   1:  PR[91,2] = PR[90,2] + 13.774;
   1:L PR[91] R[100]mm/sec CNT100;
   1:  PR[91,1] = PR[90,1] + 28.237;
   1:  PR[91,2] = PR[90,2] + 15.206;
   1:L PR[91] R[100]mm/sec CNT100;
   1:  PR[91,1] = PR[90,1] + 27.710;
   1:  PR[91,2] = PR[90,2] + 15.533;
   1:L PR[91] R[100]mm/sec CNT100;
   1:  PR[91,1] = PR[90,1] + 25.602;
   1:  PR[91,2] = PR[90,2] + 16.678;
   1:L PR[91] R[100]mm/sec CNT100;
   1:  PR[91,1] = PR[90,1] + 23.587;
   1:  PR[91,2] = PR[90,2] + 17.443;
   1:L PR[91] R[100]mm/sec CNT100;
   1:  PR[91,1] = PR[90,1] + 22.466;
   1:  PR[91,2] = PR[90,2] + 17.845;
   1:L PR[91] R[100]mm/sec CNT100;
   1:  PR[91,1] = PR[90,1] + 20.601;
   1:  PR[91,2] = PR[90,2] + 18.286;
   1:L PR[91] R[100]mm/sec CNT100;
   1:  PR[91,1] = PR[90,1] + 18.780;
   1:  PR[91,2] = PR[90,2] + 18.458;
   1:L PR[91] R[100]mm/sec CNT100;
   1:  PR[91,1] = PR[90,1] + 17.067;
   1:  PR[91,2] = PR[90,2] + 18.689;
   1:L PR[91] R[100]mm/sec CNT100;
   1:  PR[91,1] = PR[90,1] + 15.509;
   1:  PR[91,2] = PR[90,2] + 18.636;
   1:L PR[91] R[100]mm/sec CNT100;
   1:  PR[91,1] = PR[90,1] + 13.386;
   1:  PR[91,2] = PR[90,2] + 18.465;
   1:L PR[91] R[100]mm/sec CNT100;
   1:  PR[91,1] = PR[90,1] + 12.007;
   1:  PR[91,2] = PR[90,2] + 18.232;
   1:L PR[91] R[100]mm/sec CNT100;
   1:  PR[91,1] = PR[90,1] + 10.743;
   1:  PR[91,2] = PR[90,2] + 17.834;
   1:L PR[91] R[100]mm/sec CNT100;
   1:  PR[91,1] = PR[90,1] + 8.282;
   1:  PR[91,2] = PR[90,2] + 17.090;
   1:L PR[91] R[100]mm/sec CNT100;
   1:  PR[91,1] = PR[90,1] + 7.321;
   1:  PR[91,2] = PR[90,2] + 16.639;
   1:L PR[91] R[100]mm/sec CNT100;
   1:  PR[91,1] = PR[90,1] + 4.764;
   1:  PR[91,2] = PR[90,2] + 15.203;
   1:L PR[91] R[100]mm/sec CNT100;
   1:  PR[91,1] = PR[90,1] + 3.982;
   1:  PR[91,2] = PR[90,2] + 14.693;
   1:L PR[91] R[100]mm/sec CNT100;
   1:  PR[91,1] = PR[90,1] + 2.880;
   1:  PR[91,2] = PR[90,2] + 13.777;
   1:L PR[91] R[100]mm/sec CNT100;
   1:  PR[91,1] = PR[90,1] + 2.134;
   1:  PR[91,2] = PR[90,2] + 13.086;
   1:L PR[91] R[100]mm/sec CNT100;
   1:  PR[91,1] = PR[90,1] + 1.372;
   1:  PR[91,2] = PR[90,2] + 12.629;
   1:L PR[91] R[100]mm/sec CNT100;
   1:  PR[91,1] = PR[90,1] + 0.512;
   1:  PR[91,2] = PR[90,2] + 12.269;
   1:L PR[91] R[100]mm/sec CNT100;
   1:  PR[91] = PR[90];
   1:  PR[91,1] = PR[90,1] + -1.049;
   1:  PR[91,2] = PR[90,2] + 12.856;
   1:  PR[91,3] = PR[90,3] + 32.695;
   1:L PR[91] R[100]mm/sec CNT100;
   1:  PR[91,1] = PR[90,1] + -2.250;
   1:  PR[91,2] = PR[90,2] + 13.413;
   1:L PR[91] R[100]mm/sec CNT100;
   1:  PR[91,1] = PR[90,1] + -3.926;
   1:  PR[91,2] = PR[90,2] + 14.817;
   1:L PR[91] R[100]mm/sec CNT100;
   1:  PR[91,1] = PR[90,1] + -4.466;
   1:  PR[91,2] = PR[90,2] + 15.172;
   1:L PR[91] R[100]mm/sec CNT100;
   1:  PR[91,1] = PR[90,1] + -7.479;
   1:  PR[91,2] = PR[90,2] + 16.866;
   1:L PR[91] R[100]mm/sec CNT100;
   1:  PR[91,1] = PR[90,1] + -8.163;
   1:  PR[91,2] = PR[90,2] + 17.188;
   1:L PR[91] R[100]mm/sec CNT100;
   1:  PR[91,1] = PR[90,1] + -12.073;
   1:  PR[91,2] = PR[90,2] + 18.383;
   1:L PR[91] R[100]mm/sec CNT100;
   1:  PR[91,1] = PR[90,1] + -13.127;
   1:  PR[91,2] = PR[90,2] + 18.559;
   1:L PR[91] R[100]mm/sec CNT100;
   1:  PR[91,1] = PR[90,1] + -15.795;
   1:  PR[91,2] = PR[90,2] + 18.773;
   1:L PR[91] R[100]mm/sec CNT100;
   1:  PR[91,1] = PR[90,1] + -17.081;
   1:  PR[91,2] = PR[90,2] + 18.816;
   1:L PR[91] R[100]mm/sec CNT100;
   1:  PR[91,1] = PR[90,1] + -18.591;
   1:  PR[91,2] = PR[90,2] + 18.666;
   1:L PR[91] R[100]mm/sec CNT100;
   1:  PR[91,1] = PR[90,1] + -20.751;
   1:  PR[91,2] = PR[90,2] + 18.379;
   1:L PR[91] R[100]mm/sec CNT100;
   1:  PR[91,1] = PR[90,1] + -22.305;
   1:  PR[91,2] = PR[90,2] + 18.011;
   1:L PR[91] R[100]mm/sec CNT100;
   1:  PR[91,1] = PR[90,1] + -24.173;
   1:  PR[91,2] = PR[90,2] + 17.302;
   1:L PR[91] R[100]mm/sec CNT100;
   1:  PR[91,1] = PR[90,1] + -25.691;
   1:  PR[91,2] = PR[90,2] + 16.756;
   1:L PR[91] R[100]mm/sec CNT100;
   1:  PR[91,1] = PR[90,1] + -27.462;
   1:  PR[91,2] = PR[90,2] + 15.788;
   1:L PR[91] R[100]mm/sec CNT100;
   1:  PR[91,1] = PR[90,1] + -28.488;
   1:  PR[91,2] = PR[90,2] + 15.149;
   1:L PR[91] R[100]mm/sec CNT100;
   1:  PR[91,1] = PR[90,1] + -30.178;
   1:  PR[91,2] = PR[90,2] + 13.903;
   1:L PR[91] R[100]mm/sec CNT100;
   1:  PR[91,1] = PR[90,1] + -32.399;
   1:  PR[91,2] = PR[90,2] + 11.739;
   1:L PR[91] R[100]mm/sec CNT100;
   1:  PR[91,1] = PR[90,1] + -33.837;
   1:  PR[91,2] = PR[90,2] + 9.866;
   1:L PR[91] R[100]mm/sec CNT100;
   1:  PR[91,1] = PR[90,1] + -34.082;
   1:  PR[91,2] = PR[90,2] + 9.483;
   1:L PR[91] R[100]mm/sec CNT100;
   1:  PR[91,1] = PR[90,1] + -35.313;
   1:  PR[91,2] = PR[90,2] + 7.290;
   1:L PR[91] R[100]mm/sec CNT100;
   1:  PR[91,1] = PR[90,1] + -36.348;
   1:  PR[91,2] = PR[90,2] + 4.612;
   1:L PR[91] R[100]mm/sec CNT100;
   1:  PR[91,1] = PR[90,1] + -36.871;
   1:  PR[91,2] = PR[90,2] + 2.281;
   1:L PR[91] R[100]mm/sec CNT100;
   1:  PR[91,1] = PR[90,1] + -37.069;
   1:  PR[91,2] = PR[90,2] + -0.428;
   1:L PR[91] R[100]mm/sec CNT100;
   1:  PR[91,1] = PR[90,1] + -36.891;
   1:  PR[91,2] = PR[90,2] + -3.008;
   1:L PR[91] R[100]mm/sec CNT100;
   1:  PR[91,1] = PR[90,1] + -36.882;
   1:  PR[91,2] = PR[90,2] + -3.078;
   1:L PR[91] R[100]mm/sec CNT100;
   1:  PR[91,1] = PR[90,1] + -36.349;
   1:  PR[91,2] = PR[90,2] + -5.456;
   1:L PR[91] R[100]mm/sec CNT100;
   1:  PR[91,1] = PR[90,1] + -35.394;
   1:  PR[91,2] = PR[90,2] + -7.905;
   1:L PR[91] R[100]mm/sec CNT100;
   1:  PR[91,1] = PR[90,1] + -35.303;
   1:  PR[91,2] = PR[90,2] + -8.156;
   1:L PR[91] R[100]mm/sec CNT100;
   1:  PR[91,1] = PR[90,1] + -34.083;
   1:  PR[91,2] = PR[90,2] + -10.331;
   1:L PR[91] R[100]mm/sec CNT100;
   1:  PR[91,1] = PR[90,1] + -33.837;
   1:  PR[91,2] = PR[90,2] + -10.713;
   1:L PR[91] R[100]mm/sec CNT100;
   1:  PR[91,1] = PR[90,1] + -32.399;
   1:  PR[91,2] = PR[90,2] + -12.586;
   1:L PR[91] R[100]mm/sec CNT100;
   1:  PR[91,1] = PR[90,1] + -30.178;
   1:  PR[91,2] = PR[90,2] + -14.750;
   1:L PR[91] R[100]mm/sec CNT100;
   1:  PR[91,1] = PR[90,1] + -28.488;
   1:  PR[91,2] = PR[90,2] + -15.996;
   1:L PR[91] R[100]mm/sec CNT100;
   1:  PR[91,1] = PR[90,1] + -27.462;
   1:  PR[91,2] = PR[90,2] + -16.636;
   1:L PR[91] R[100]mm/sec CNT100;
   1:  PR[91,1] = PR[90,1] + -25.670;
   1:  PR[91,2] = PR[90,2] + -17.614;
   1:L PR[91] R[100]mm/sec CNT100;
   1:  PR[91,1] = PR[90,1] + -23.969;
   1:  PR[91,2] = PR[90,2] + -18.263;
   1:L PR[91] R[100]mm/sec CNT100;
   1:  PR[91,1] = PR[90,1] + -22.326;
   1:  PR[91,2] = PR[90,2] + -18.853;
   1:L PR[91] R[100]mm/sec CNT100;
   1:  PR[91,1] = PR[90,1] + -20.794;
   1:  PR[91,2] = PR[90,2] + -19.216;
   1:L PR[91] R[100]mm/sec CNT100;
   1:  PR[91,1] = PR[90,1] + -19.268;
   1:  PR[91,2] = PR[90,2] + -19.362;
   1:L PR[91] R[100]mm/sec CNT100;
   1:  PR[91,1] = PR[90,1] + -17.039;
   1:  PR[91,2] = PR[90,2] + -19.662;
   1:L PR[91] R[100]mm/sec CNT100;
   1:  PR[91,1] = PR[90,1] + -15.794;
   1:  PR[91,2] = PR[90,2] + -19.620;
   1:L PR[91] R[100]mm/sec CNT100;
   1:  PR[91,1] = PR[90,1] + -13.127;
   1:  PR[91,2] = PR[90,2] + -19.407;
   1:L PR[91] R[100]mm/sec CNT100;
   1:  PR[91,1] = PR[90,1] + -12.073;
   1:  PR[91,2] = PR[90,2] + -19.230;
   1:L PR[91] R[100]mm/sec CNT100;
   1:  PR[91,1] = PR[90,1] + -8.162;
   1:  PR[91,2] = PR[90,2] + -18.035;
   1:L PR[91] R[100]mm/sec CNT100;
   1:  PR[91,1] = PR[90,1] + -7.479;
   1:  PR[91,2] = PR[90,2] + -17.714;
   1:L PR[91] R[100]mm/sec CNT100;
   1:  PR[91,1] = PR[90,1] + -4.462;
   1:  PR[91,2] = PR[90,2] + -16.017;
   1:L PR[91] R[100]mm/sec CNT100;
   1:  PR[91,1] = PR[90,1] + -3.943;
   1:  PR[91,2] = PR[90,2] + -15.678;
   1:L PR[91] R[100]mm/sec CNT100;
   1:  PR[91,1] = PR[90,1] + -2.534;
   1:  PR[91,2] = PR[90,2] + -14.508;
   1:L PR[91] R[100]mm/sec CNT100;
   1:  PR[91,1] = PR[90,1] + -2.341;
   1:  PR[91,2] = PR[90,2] + -14.431;
   1:L PR[91] R[100]mm/sec CNT100;
   1:  PR[91,1] = PR[90,1] + -0.931;
   1:  PR[91,2] = PR[90,2] + -13.498;
   1:L PR[91] R[100]mm/sec CNT100;
   1:  PR[91,1] = PR[90,1] + 0.392;
   1:  PR[91,2] = PR[90,2] + -13.866;
   1:L PR[91] R[100]mm/sec CNT100;
   1:  PR[91,1] = PR[90,1] + 1.089;
   1:  PR[91,2] = PR[90,2] + -13.867;
   1:L PR[91] R[100]mm/sec CNT100;
   1:  PR[91,1] = PR[90,1] + 2.270;
   1:  PR[91,2] = PR[90,2] + -14.689;
   1:L PR[91] R[100]mm/sec CNT100;
   1:  PR[91,1] = PR[90,1] + 3.439;
   1:  PR[91,2] = PR[90,2] + -15.663;
   1:L PR[91] R[100]mm/sec CNT100;
   1:  PR[91,1] = PR[90,1] + 3.981;
   1:  PR[91,2] = PR[90,2] + -16.019;
   1:L PR[91] R[100]mm/sec CNT100;
   1:  PR[91,1] = PR[90,1] + 6.994;
   1:  PR[91,2] = PR[90,2] + -17.712;
   1:L PR[91] R[100]mm/sec CNT100;
   1:  PR[91,1] = PR[90,1] + 7.674;
   1:  PR[91,2] = PR[90,2] + -18.031;
   1:L PR[91] R[100]mm/sec CNT100;
   1:  PR[91,1] = PR[90,1] + 11.589;
   1:  PR[91,2] = PR[90,2] + -19.228;
   1:L PR[91] R[100]mm/sec CNT100;
   1:  PR[91,1] = PR[90,1] + 12.644;
   1:  PR[91,2] = PR[90,2] + -19.406;
   1:L PR[91] R[100]mm/sec CNT100;
   1:  PR[91,1] = PR[90,1] + 15.311;
   1:  PR[91,2] = PR[90,2] + -19.621;
   1:L PR[91] R[100]mm/sec CNT100;
   1:  PR[91,1] = PR[90,1] + 16.592;
   1:  PR[91,2] = PR[90,2] + -19.664;
   1:L PR[91] R[100]mm/sec CNT100;
   1:  PR[91,1] = PR[90,1] + 18.093;
   1:  PR[91,2] = PR[90,2] + -19.516;
   1:L PR[91] R[100]mm/sec CNT100;
   1:  PR[91,1] = PR[90,1] + 20.254;
   1:  PR[91,2] = PR[90,2] + -19.229;
   1:L PR[91] R[100]mm/sec CNT100;
   1:  PR[91,1] = PR[90,1] + 21.807;
   1:  PR[91,2] = PR[90,2] + -18.862;
   1:L PR[91] R[100]mm/sec CNT100;
   1:  PR[91,1] = PR[90,1] + 23.679;
   1:  PR[91,2] = PR[90,2] + -18.155;
   1:L PR[91] R[100]mm/sec CNT100;
   1:  PR[91,1] = PR[90,1] + 25.198;
   1:  PR[91,2] = PR[90,2] + -17.609;
   1:L PR[91] R[100]mm/sec CNT100;
   1:  PR[91,1] = PR[90,1] + 26.962;
   1:  PR[91,2] = PR[90,2] + -16.651;
   1:L PR[91] R[100]mm/sec CNT100;
   1:  PR[91,1] = PR[90,1] + 27.990;
   1:  PR[91,2] = PR[90,2] + -16.012;
   1:L PR[91] R[100]mm/sec CNT100;
   1:  PR[91,1] = PR[90,1] + 29.661;
   1:  PR[91,2] = PR[90,2] + -14.785;
   1:L PR[91] R[100]mm/sec CNT100;
   1:  PR[91,1] = PR[90,1] + 31.880;
   1:  PR[91,2] = PR[90,2] + -12.625;
   1:L PR[91] R[100]mm/sec CNT100;
   1:  PR[91,1] = PR[90,1] + 33.333;
   1:  PR[91,2] = PR[90,2] + -10.737;
   1:L PR[91] R[100]mm/sec CNT100;
   1:  PR[91,1] = PR[90,1] + 33.582;
   1:  PR[91,2] = PR[90,2] + -10.350;
   1:L PR[91] R[100]mm/sec CNT100;
   1:  PR[91,1] = PR[90,1] + 34.825;
   1:  PR[91,2] = PR[90,2] + -8.156;
   1:L PR[91] R[100]mm/sec CNT100;
   1:  PR[91,1] = PR[90,1] + 35.854;
   1:  PR[91,2] = PR[90,2] + -5.527;
   1:L PR[91] R[100]mm/sec CNT100;
   1:  PR[91,1] = PR[90,1] + 36.380;
   1:  PR[91,2] = PR[90,2] + -3.215;
   1:L PR[91] R[100]mm/sec CNT100;
   1:  PR[91,1] = PR[90,1] + 36.589;
   1:  PR[91,2] = PR[90,2] + -0.419;
   1:L PR[91] R[100]mm/sec CNT100;
   1:  PR[91,1] = PR[90,1] + 36.399;
   1:  PR[91,2] = PR[90,2] + 2.249;
   1:L PR[91] R[100]mm/sec CNT100;
   1:  PR[91,1] = PR[90,1] + 36.391;
   1:  PR[91,2] = PR[90,2] + 2.320;
   1:L PR[91] R[100]mm/sec CNT100;
   1:  PR[91,1] = PR[90,1] + 35.854;
   1:  PR[91,2] = PR[90,2] + 4.680;
   1:L PR[91] R[100]mm/sec CNT100;
   1:  PR[91,1] = PR[90,1] + 34.825;
   1:  PR[91,2] = PR[90,2] + 7.309;
   1:L PR[91] R[100]mm/sec CNT100;
   1:  PR[91,1] = PR[90,1] + 33.582;
   1:  PR[91,2] = PR[90,2] + 9.503;
   1:L PR[91] R[100]mm/sec CNT100;
   1:  PR[91,1] = PR[90,1] + 33.334;
   1:  PR[91,2] = PR[90,2] + 9.890;
   1:L PR[91] R[100]mm/sec CNT100;
   1:  PR[91,1] = PR[90,1] + 31.880;
   1:  PR[91,2] = PR[90,2] + 11.778;
   1:L PR[91] R[100]mm/sec CNT100;
   1:  PR[91,1] = PR[90,1] + 29.661;
   1:  PR[91,2] = PR[90,2] + 13.938;
   1:L PR[91] R[100]mm/sec CNT100;
   1:  PR[91,1] = PR[90,1] + 27.990;
   1:  PR[91,2] = PR[90,2] + 15.164;
   1:L PR[91] R[100]mm/sec CNT100;
   1:  PR[91,1] = PR[90,1] + 26.962;
   1:  PR[91,2] = PR[90,2] + 15.804;
   1:L PR[91] R[100]mm/sec CNT100;
   1:  PR[91,1] = PR[90,1] + 25.180;
   1:  PR[91,2] = PR[90,2] + 16.772;
   1:L PR[91] R[100]mm/sec CNT100;
   1:  PR[91,1] = PR[90,1] + 23.473;
   1:  PR[91,2] = PR[90,2] + 17.420;
   1:L PR[91] R[100]mm/sec CNT100;
   1:  PR[91,1] = PR[90,1] + 21.827;
   1:  PR[91,2] = PR[90,2] + 18.010;
   1:L PR[91] R[100]mm/sec CNT100;
   1:  PR[91,1] = PR[90,1] + 20.298;
   1:  PR[91,2] = PR[90,2] + 18.371;
   1:L PR[91] R[100]mm/sec CNT100;
   1:  PR[91,1] = PR[90,1] + 18.779;
   1:  PR[91,2] = PR[90,2] + 18.515;
   1:L PR[91] R[100]mm/sec CNT100;
   1:  PR[91,1] = PR[90,1] + 16.549;
   1:  PR[91,2] = PR[90,2] + 18.815;
   1:L PR[91] R[100]mm/sec CNT100;
   1:  PR[91,1] = PR[90,1] + 15.311;
   1:  PR[91,2] = PR[90,2] + 18.773;
   1:L PR[91] R[100]mm/sec CNT100;
   1:  PR[91,1] = PR[90,1] + 12.644;
   1:  PR[91,2] = PR[90,2] + 18.559;
   1:L PR[91] R[100]mm/sec CNT100;
   1:  PR[91,1] = PR[90,1] + 11.589;
   1:  PR[91,2] = PR[90,2] + 18.381;
   1:L PR[91] R[100]mm/sec CNT100;
   1:  PR[91,1] = PR[90,1] + 7.675;
   1:  PR[91,2] = PR[90,2] + 17.184;
   1:L PR[91] R[100]mm/sec CNT100;
   1:  PR[91,1] = PR[90,1] + 6.995;
   1:  PR[91,2] = PR[90,2] + 16.865;
   1:L PR[91] R[100]mm/sec CNT100;
   1:  PR[91,1] = PR[90,1] + 3.979;
   1:  PR[91,2] = PR[90,2] + 15.171;
   1:L PR[91] R[100]mm/sec CNT100;
   1:  PR[91,1] = PR[90,1] + 3.466;
   1:  PR[91,2] = PR[90,2] + 14.837;
   1:L PR[91] R[100]mm/sec CNT100;
   1:  PR[91,1] = PR[90,1] + 2.160;
   1:  PR[91,2] = PR[90,2] + 13.750;
   1:L PR[91] R[100]mm/sec CNT100;
   1:  PR[91,1] = PR[90,1] + 2.126;
   1:  PR[91,2] = PR[90,2] + 13.732;
   1:L PR[91] R[100]mm/sec CNT100;
   1:  PR[91,1] = PR[90,1] + 1.996;
   1:  PR[91,2] = PR[90,2] + 13.616;
   1:L PR[91] R[100]mm/sec CNT100;
   1:  PR[91,1] = PR[90,1] + 1.420;
   1:  PR[91,2] = PR[90,2] + 13.271;
   1:L PR[91] R[100]mm/sec CNT100;
   1:  PR[91,1] = PR[90,1] + 0.432;
   1:  PR[91,2] = PR[90,2] + 12.857;
   1:L PR[91] R[100]mm/sec CNT100;
   1:  PR[91] = PR[90];
   1:  PR[91,1] = PR[90,1] + -1.001;
   1:  PR[91,2] = PR[90,2] + 13.445;
   1:  PR[91,3] = PR[90,3] + 33.995;
   1:L PR[91] R[100]mm/sec CNT100;
   1:  PR[91,1] = PR[90,1] + -2.346;
   1:  PR[91,2] = PR[90,2] + 14.068;
   1:L PR[91] R[100]mm/sec CNT100;
   1:  PR[91,1] = PR[90,1] + -3.412;
   1:  PR[91,2] = PR[90,2] + 14.963;
   1:L PR[91] R[100]mm/sec CNT100;
   1:  PR[91,1] = PR[90,1] + -3.683;
   1:  PR[91,2] = PR[90,2] + 15.142;
   1:L PR[91] R[100]mm/sec CNT100;
   1:  PR[91,1] = PR[90,1] + -7.153;
   1:  PR[91,2] = PR[90,2] + 17.092;
   1:L PR[91] R[100]mm/sec CNT100;
   1:  PR[91,1] = PR[90,1] + -7.551;
   1:  PR[91,2] = PR[90,2] + 17.279;
   1:L PR[91] R[100]mm/sec CNT100;
   1:  PR[91,1] = PR[90,1] + -11.664;
   1:  PR[91,2] = PR[90,2] + 18.532;
   1:L PR[91] R[100]mm/sec CNT100;
   1:  PR[91,1] = PR[90,1] + -12.385;
   1:  PR[91,2] = PR[90,2] + 18.653;
   1:L PR[91] R[100]mm/sec CNT100;
   1:  PR[91,1] = PR[90,1] + -15.596;
   1:  PR[91,2] = PR[90,2] + 18.911;
   1:L PR[91] R[100]mm/sec CNT100;
   1:  PR[91,1] = PR[90,1] + -16.561;
   1:  PR[91,2] = PR[90,2] + 18.943;
   1:L PR[91] R[100]mm/sec CNT100;
   1:  PR[91,1] = PR[90,1] + -17.706;
   1:  PR[91,2] = PR[90,2] + 18.829;
   1:L PR[91] R[100]mm/sec CNT100;
   1:  PR[91,1] = PR[90,1] + -20.446;
   1:  PR[91,2] = PR[90,2] + 18.465;
   1:L PR[91] R[100]mm/sec CNT100;
   1:  PR[91,1] = PR[90,1] + -21.662;
   1:  PR[91,2] = PR[90,2] + 18.177;
   1:L PR[91] R[100]mm/sec CNT100;
   1:  PR[91,1] = PR[90,1] + -23.162;
   1:  PR[91,2] = PR[90,2] + 17.608;
   1:L PR[91] R[100]mm/sec CNT100;
   1:  PR[91,1] = PR[90,1] + -25.266;
   1:  PR[91,2] = PR[90,2] + 16.850;
   1:L PR[91] R[100]mm/sec CNT100;
   1:  PR[91,1] = PR[90,1] + -26.711;
   1:  PR[91,2] = PR[90,2] + 16.061;
   1:L PR[91] R[100]mm/sec CNT100;
   1:  PR[91,1] = PR[90,1] + -28.239;
   1:  PR[91,2] = PR[90,2] + 15.109;
   1:L PR[91] R[100]mm/sec CNT100;
   1:  PR[91,1] = PR[90,1] + -29.647;
   1:  PR[91,2] = PR[90,2] + 14.071;
   1:L PR[91] R[100]mm/sec CNT100;
   1:  PR[91,1] = PR[90,1] + -32.034;
   1:  PR[91,2] = PR[90,2] + 11.742;
   1:L PR[91] R[100]mm/sec CNT100;
   1:  PR[91,1] = PR[90,1] + -33.251;
   1:  PR[91,2] = PR[90,2] + 10.156;
   1:L PR[91] R[100]mm/sec CNT100;
   1:  PR[91,1] = PR[90,1] + -33.817;
   1:  PR[91,2] = PR[90,2] + 9.276;
   1:L PR[91] R[100]mm/sec CNT100;
   1:  PR[91,1] = PR[90,1] + -34.872;
   1:  PR[91,2] = PR[90,2] + 7.394;
   1:L PR[91] R[100]mm/sec CNT100;
   1:  PR[91,1] = PR[90,1] + -35.714;
   1:  PR[91,2] = PR[90,2] + 5.229;
   1:L PR[91] R[100]mm/sec CNT100;
   1:  PR[91,1] = PR[90,1] + -35.969;
   1:  PR[91,2] = PR[90,2] + 4.534;
   1:L PR[91] R[100]mm/sec CNT100;
   1:  PR[91,1] = PR[90,1] + -36.419;
   1:  PR[91,2] = PR[90,2] + 2.526;
   1:L PR[91] R[100]mm/sec CNT100;
   1:  PR[91,1] = PR[90,1] + -36.581;
   1:  PR[91,2] = PR[90,2] + 0.186;
   1:L PR[91] R[100]mm/sec CNT100;
   1:  PR[91,1] = PR[90,1] + -36.658;
   1:  PR[91,2] = PR[90,2] + -0.479;
   1:L PR[91] R[100]mm/sec CNT100;
   1:  PR[91,1] = PR[90,1] + -36.508;
   1:  PR[91,2] = PR[90,2] + -2.658;
   1:L PR[91] R[100]mm/sec CNT100;
   1:  PR[91,1] = PR[90,1] + -36.431;
   1:  PR[91,2] = PR[90,2] + -3.319;
   1:L PR[91] R[100]mm/sec CNT100;
   1:  PR[91,1] = PR[90,1] + -35.974;
   1:  PR[91,2] = PR[90,2] + -5.357;
   1:L PR[91] R[100]mm/sec CNT100;
   1:  PR[91,1] = PR[90,1] + -35.148;
   1:  PR[91,2] = PR[90,2] + -7.478;
   1:L PR[91] R[100]mm/sec CNT100;
   1:  PR[91,1] = PR[90,1] + -34.860;
   1:  PR[91,2] = PR[90,2] + -8.263;
   1:L PR[91] R[100]mm/sec CNT100;
   1:  PR[91,1] = PR[90,1] + -33.817;
   1:  PR[91,2] = PR[90,2] + -10.123;
   1:L PR[91] R[100]mm/sec CNT100;
   1:  PR[91,1] = PR[90,1] + -33.251;
   1:  PR[91,2] = PR[90,2] + -11.004;
   1:L PR[91] R[100]mm/sec CNT100;
   1:  PR[91,1] = PR[90,1] + -32.034;
   1:  PR[91,2] = PR[90,2] + -12.589;
   1:L PR[91] R[100]mm/sec CNT100;
   1:  PR[91,1] = PR[90,1] + -29.647;
   1:  PR[91,2] = PR[90,2] + -14.919;
   1:L PR[91] R[100]mm/sec CNT100;
   1:  PR[91,1] = PR[90,1] + -28.239;
   1:  PR[91,2] = PR[90,2] + -15.957;
   1:L PR[91] R[100]mm/sec CNT100;
   1:  PR[91,1] = PR[90,1] + -26.711;
   1:  PR[91,2] = PR[90,2] + -16.908;
   1:L PR[91] R[100]mm/sec CNT100;
   1:  PR[91,1] = PR[90,1] + -25.246;
   1:  PR[91,2] = PR[90,2] + -17.709;
   1:L PR[91] R[100]mm/sec CNT100;
   1:  PR[91,1] = PR[90,1] + -23.852;
   1:  PR[91,2] = PR[90,2] + -18.241;
   1:L PR[91] R[100]mm/sec CNT100;
   1:  PR[91,1] = PR[90,1] + -21.683;
   1:  PR[91,2] = PR[90,2] + -19.019;
   1:L PR[91] R[100]mm/sec CNT100;
   1:  PR[91,1] = PR[90,1] + -20.489;
   1:  PR[91,2] = PR[90,2] + -19.302;
   1:L PR[91] R[100]mm/sec CNT100;
   1:  PR[91,1] = PR[90,1] + -19.266;
   1:  PR[91,2] = PR[90,2] + -19.419;
   1:L PR[91] R[100]mm/sec CNT100;
   1:  PR[91,1] = PR[90,1] + -16.519;
   1:  PR[91,2] = PR[90,2] + -19.789;
   1:L PR[91] R[100]mm/sec CNT100;
   1:  PR[91,1] = PR[90,1] + -15.596;
   1:  PR[91,2] = PR[90,2] + -19.758;
   1:L PR[91] R[100]mm/sec CNT100;
   1:  PR[91,1] = PR[90,1] + -12.385;
   1:  PR[91,2] = PR[90,2] + -19.501;
   1:L PR[91] R[100]mm/sec CNT100;
   1:  PR[91,1] = PR[90,1] + -11.663;
   1:  PR[91,2] = PR[90,2] + -19.380;
   1:L PR[91] R[100]mm/sec CNT100;
   1:  PR[91,1] = PR[90,1] + -7.550;
   1:  PR[91,2] = PR[90,2] + -18.126;
   1:L PR[91] R[100]mm/sec CNT100;
   1:  PR[91,1] = PR[90,1] + -7.153;
   1:  PR[91,2] = PR[90,2] + -17.940;
   1:L PR[91] R[100]mm/sec CNT100;
   1:  PR[91,1] = PR[90,1] + -3.677;
   1:  PR[91,2] = PR[90,2] + -15.985;
   1:L PR[91] R[100]mm/sec CNT100;
   1:  PR[91,1] = PR[90,1] + -3.430;
   1:  PR[91,2] = PR[90,2] + -15.824;
   1:L PR[91] R[100]mm/sec CNT100;
   1:  PR[91,1] = PR[90,1] + -2.496;
   1:  PR[91,2] = PR[90,2] + -15.049;
   1:L PR[91] R[100]mm/sec CNT100;
   1:  PR[91,1] = PR[90,1] + -2.102;
   1:  PR[91,2] = PR[90,2] + -14.893;
   1:L PR[91] R[100]mm/sec CNT100;
   1:  PR[91,1] = PR[90,1] + -0.884;
   1:  PR[91,2] = PR[90,2] + -14.086;
   1:L PR[91] R[100]mm/sec CNT100;
   1:  PR[91,1] = PR[90,1] + 0.632;
   1:  PR[91,2] = PR[90,2] + -14.508;
   1:L PR[91] R[100]mm/sec CNT100;
   1:  PR[91,1] = PR[90,1] + 1.161;
   1:  PR[91,2] = PR[90,2] + -14.509;
   1:L PR[91] R[100]mm/sec CNT100;
   1:  PR[91,1] = PR[90,1] + 1.777;
   1:  PR[91,2] = PR[90,2] + -14.955;
   1:L PR[91] R[100]mm/sec CNT100;
   1:  PR[91,1] = PR[90,1] + 2.122;
   1:  PR[91,2] = PR[90,2] + -15.139;
   1:L PR[91] R[100]mm/sec CNT100;
   1:  PR[91,1] = PR[90,1] + 2.923;
   1:  PR[91,2] = PR[90,2] + -15.806;
   1:L PR[91] R[100]mm/sec CNT100;
   1:  PR[91,1] = PR[90,1] + 3.199;
   1:  PR[91,2] = PR[90,2] + -15.988;
   1:L PR[91] R[100]mm/sec CNT100;
   1:  PR[91,1] = PR[90,1] + 6.668;
   1:  PR[91,2] = PR[90,2] + -17.938;
   1:L PR[91] R[100]mm/sec CNT100;
   1:  PR[91,1] = PR[90,1] + 7.063;
   1:  PR[91,2] = PR[90,2] + -18.123;
   1:L PR[91] R[100]mm/sec CNT100;
   1:  PR[91,1] = PR[90,1] + 11.180;
   1:  PR[91,2] = PR[90,2] + -19.378;
   1:L PR[91] R[100]mm/sec CNT100;
   1:  PR[91,1] = PR[90,1] + 11.902;
   1:  PR[91,2] = PR[90,2] + -19.500;
   1:L PR[91] R[100]mm/sec CNT100;
   1:  PR[91,1] = PR[90,1] + 15.113;
   1:  PR[91,2] = PR[90,2] + -19.758;
   1:L PR[91] R[100]mm/sec CNT100;
   1:  PR[91,1] = PR[90,1] + 16.074;
   1:  PR[91,2] = PR[90,2] + -19.791;
   1:L PR[91] R[100]mm/sec CNT100;
   1:  PR[91,1] = PR[90,1] + 17.211;
   1:  PR[91,2] = PR[90,2] + -19.679;
   1:L PR[91] R[100]mm/sec CNT100;
   1:  PR[91,1] = PR[90,1] + 19.951;
   1:  PR[91,2] = PR[90,2] + -19.315;
   1:L PR[91] R[100]mm/sec CNT100;
   1:  PR[91,1] = PR[90,1] + 21.167;
   1:  PR[91,2] = PR[90,2] + -19.027;
   1:L PR[91] R[100]mm/sec CNT100;
   1:  PR[91,1] = PR[90,1] + 22.670;
   1:  PR[91,2] = PR[90,2] + -18.460;
   1:L PR[91] R[100]mm/sec CNT100;
   1:  PR[91,1] = PR[90,1] + 24.776;
   1:  PR[91,2] = PR[90,2] + -17.702;
   1:L PR[91] R[100]mm/sec CNT100;
   1:  PR[91,1] = PR[90,1] + 26.215;
   1:  PR[91,2] = PR[90,2] + -16.921;
   1:L PR[91] R[100]mm/sec CNT100;
   1:  PR[91,1] = PR[90,1] + 27.744;
   1:  PR[91,2] = PR[90,2] + -15.970;
   1:L PR[91] R[100]mm/sec CNT100;
   1:  PR[91,1] = PR[90,1] + 29.135;
   1:  PR[91,2] = PR[90,2] + -14.949;
   1:L PR[91] R[100]mm/sec CNT100;
   1:  PR[91,1] = PR[90,1] + 31.521;
   1:  PR[91,2] = PR[90,2] + -12.622;
   1:L PR[91] R[100]mm/sec CNT100;
   1:  PR[91,1] = PR[90,1] + 32.751;
   1:  PR[91,2] = PR[90,2] + -11.023;
   1:L PR[91] R[100]mm/sec CNT100;
   1:  PR[91,1] = PR[90,1] + 33.319;
   1:  PR[91,2] = PR[90,2] + -10.139;
   1:L PR[91] R[100]mm/sec CNT100;
   1:  PR[91,1] = PR[90,1] + 34.386;
   1:  PR[91,2] = PR[90,2] + -8.257;
   1:L PR[91] R[100]mm/sec CNT100;
   1:  PR[91,1] = PR[90,1] + 35.221;
   1:  PR[91,2] = PR[90,2] + -6.137;
   1:L PR[91] R[100]mm/sec CNT100;
   1:  PR[91,1] = PR[90,1] + 35.476;
   1:  PR[91,2] = PR[90,2] + -5.445;
   1:L PR[91] R[100]mm/sec CNT100;
   1:  PR[91,1] = PR[90,1] + 35.930;
   1:  PR[91,2] = PR[90,2] + -3.450;
   1:L PR[91] R[100]mm/sec CNT100;
   1:  PR[91,1] = PR[90,1] + 36.102;
   1:  PR[91,2] = PR[90,2] + -1.034;
   1:L PR[91] R[100]mm/sec CNT100;
   1:  PR[91,1] = PR[90,1] + 36.178;
   1:  PR[91,2] = PR[90,2] + -0.371;
   1:L PR[91] R[100]mm/sec CNT100;
   1:  PR[91,1] = PR[90,1] + 36.018;
   1:  PR[91,2] = PR[90,2] + 1.888;
   1:L PR[91] R[100]mm/sec CNT100;
   1:  PR[91,1] = PR[90,1] + 35.941;
   1:  PR[91,2] = PR[90,2] + 2.552;
   1:L PR[91] R[100]mm/sec CNT100;
   1:  PR[91,1] = PR[90,1] + 35.482;
   1:  PR[91,2] = PR[90,2] + 4.570;
   1:L PR[91] R[100]mm/sec CNT100;
   1:  PR[91,1] = PR[90,1] + 34.659;
   1:  PR[91,2] = PR[90,2] + 6.651;
   1:L PR[91] R[100]mm/sec CNT100;
   1:  PR[91,1] = PR[90,1] + 34.372;
   1:  PR[91,2] = PR[90,2] + 7.434;
   1:L PR[91] R[100]mm/sec CNT100;
   1:  PR[91,1] = PR[90,1] + 33.319;
   1:  PR[91,2] = PR[90,2] + 9.292;
   1:L PR[91] R[100]mm/sec CNT100;
   1:  PR[91,1] = PR[90,1] + 32.751;
   1:  PR[91,2] = PR[90,2] + 10.176;
   1:L PR[91] R[100]mm/sec CNT100;
   1:  PR[91,1] = PR[90,1] + 31.521;
   1:  PR[91,2] = PR[90,2] + 11.774;
   1:L PR[91] R[100]mm/sec CNT100;
   1:  PR[91,1] = PR[90,1] + 29.135;
   1:  PR[91,2] = PR[90,2] + 14.102;
   1:L PR[91] R[100]mm/sec CNT100;
   1:  PR[91,1] = PR[90,1] + 27.744;
   1:  PR[91,2] = PR[90,2] + 15.123;
   1:L PR[91] R[100]mm/sec CNT100;
   1:  PR[91,1] = PR[90,1] + 26.215;
   1:  PR[91,2] = PR[90,2] + 16.074;
   1:L PR[91] R[100]mm/sec CNT100;
   1:  PR[91,1] = PR[90,1] + 24.757;
   1:  PR[91,2] = PR[90,2] + 16.865;
   1:L PR[91] R[100]mm/sec CNT100;
   1:  PR[91,1] = PR[90,1] + 23.357;
   1:  PR[91,2] = PR[90,2] + 17.397;
   1:L PR[91] R[100]mm/sec CNT100;
   1:  PR[91,1] = PR[90,1] + 21.187;
   1:  PR[91,2] = PR[90,2] + 18.175;
   1:L PR[91] R[100]mm/sec CNT100;
   1:  PR[91,1] = PR[90,1] + 19.996;
   1:  PR[91,2] = PR[90,2] + 18.457;
   1:L PR[91] R[100]mm/sec CNT100;
   1:  PR[91,1] = PR[90,1] + 18.779;
   1:  PR[91,2] = PR[90,2] + 18.572;
   1:L PR[91] R[100]mm/sec CNT100;
   1:  PR[91,1] = PR[90,1] + 16.030;
   1:  PR[91,2] = PR[90,2] + 18.942;
   1:L PR[91] R[100]mm/sec CNT100;
   1:  PR[91,1] = PR[90,1] + 15.113;
   1:  PR[91,2] = PR[90,2] + 18.911;
   1:L PR[91] R[100]mm/sec CNT100;
   1:  PR[91,1] = PR[90,1] + 11.902;
   1:  PR[91,2] = PR[90,2] + 18.652;
   1:L PR[91] R[100]mm/sec CNT100;
   1:  PR[91,1] = PR[90,1] + 11.180;
   1:  PR[91,2] = PR[90,2] + 18.531;
   1:L PR[91] R[100]mm/sec CNT100;
   1:  PR[91,1] = PR[90,1] + 7.063;
   1:  PR[91,2] = PR[90,2] + 17.276;
   1:L PR[91] R[100]mm/sec CNT100;
   1:  PR[91,1] = PR[90,1] + 6.668;
   1:  PR[91,2] = PR[90,2] + 17.090;
   1:L PR[91] R[100]mm/sec CNT100;
   1:  PR[91,1] = PR[90,1] + 3.193;
   1:  PR[91,2] = PR[90,2] + 15.138;
   1:L PR[91] R[100]mm/sec CNT100;
   1:  PR[91,1] = PR[90,1] + 2.951;
   1:  PR[91,2] = PR[90,2] + 14.980;
   1:L PR[91] R[100]mm/sec CNT100;
   1:  PR[91,1] = PR[90,1] + 2.120;
   1:  PR[91,2] = PR[90,2] + 14.290;
   1:L PR[91] R[100]mm/sec CNT100;
   1:  PR[91,1] = PR[90,1] + 1.777;
   1:  PR[91,2] = PR[90,2] + 14.107;
   1:L PR[91] R[100]mm/sec CNT100;
   1:  PR[91,1] = PR[90,1] + 1.564;
   1:  PR[91,2] = PR[90,2] + 13.954;
   1:L PR[91] R[100]mm/sec CNT100;
   1:  PR[91,1] = PR[90,1] + 0.352;
   1:  PR[91,2] = PR[90,2] + 13.446;
   1:L PR[91] R[100]mm/sec CNT100;
   1:  PR[91] = PR[90];
   1:  PR[91,1] = PR[90,1] + -0.954;
   1:  PR[91,2] = PR[90,2] + 14.033;
   1:  PR[91,3] = PR[90,3] + 35.295;
   1:L PR[91] R[100]mm/sec CNT100;
   1:  PR[91,1] = PR[90,1] + -2.445;
   1:  PR[91,2] = PR[90,2] + 14.724;
   1:L PR[91] R[100]mm/sec CNT100;
   1:  PR[91,1] = PR[90,1] + -2.907;
   1:  PR[91,2] = PR[90,2] + 15.114;
   1:L PR[91] R[100]mm/sec CNT100;
   1:  PR[91,1] = PR[90,1] + -6.827;
   1:  PR[91,2] = PR[90,2] + 17.318;
   1:L PR[91] R[100]mm/sec CNT100;
   1:  PR[91,1] = PR[90,1] + -6.939;
   1:  PR[91,2] = PR[90,2] + 17.371;
   1:L PR[91] R[100]mm/sec CNT100;
   1:  PR[91,1] = PR[90,1] + -11.254;
   1:  PR[91,2] = PR[90,2] + 18.682;
   1:L PR[91] R[100]mm/sec CNT100;
   1:  PR[91,1] = PR[90,1] + -11.643;
   1:  PR[91,2] = PR[90,2] + 18.747;
   1:L PR[91] R[100]mm/sec CNT100;
   1:  PR[91,1] = PR[90,1] + -15.398;
   1:  PR[91,2] = PR[90,2] + 19.048;
   1:L PR[91] R[100]mm/sec CNT100;
   1:  PR[91,1] = PR[90,1] + -16.041;
   1:  PR[91,2] = PR[90,2] + 19.070;
   1:L PR[91] R[100]mm/sec CNT100;
   1:  PR[91,1] = PR[90,1] + -16.820;
   1:  PR[91,2] = PR[90,2] + 18.992;
   1:L PR[91] R[100]mm/sec CNT100;
   1:  PR[91,1] = PR[90,1] + -20.140;
   1:  PR[91,2] = PR[90,2] + 18.551;
   1:L PR[91] R[100]mm/sec CNT100;
   1:  PR[91,1] = PR[90,1] + -21.020;
   1:  PR[91,2] = PR[90,2] + 18.342;
   1:L PR[91] R[100]mm/sec CNT100;
   1:  PR[91,1] = PR[90,1] + -22.150;
   1:  PR[91,2] = PR[90,2] + 17.913;
   1:L PR[91] R[100]mm/sec CNT100;
   1:  PR[91,1] = PR[90,1] + -24.841;
   1:  PR[91,2] = PR[90,2] + 16.945;
   1:L PR[91] R[100]mm/sec CNT100;
   1:  PR[91,1] = PR[90,1] + -25.960;
   1:  PR[91,2] = PR[90,2] + 16.334;
   1:L PR[91] R[100]mm/sec CNT100;
   1:  PR[91,1] = PR[90,1] + -27.990;
   1:  PR[91,2] = PR[90,2] + 15.069;
   1:L PR[91] R[100]mm/sec CNT100;
   1:  PR[91,1] = PR[90,1] + -29.115;
   1:  PR[91,2] = PR[90,2] + 14.240;
   1:L PR[91] R[100]mm/sec CNT100;
   1:  PR[91,1] = PR[90,1] + -31.670;
   1:  PR[91,2] = PR[90,2] + 11.744;
   1:L PR[91] R[100]mm/sec CNT100;
   1:  PR[91,1] = PR[90,1] + -32.666;
   1:  PR[91,2] = PR[90,2] + 10.447;
   1:L PR[91] R[100]mm/sec CNT100;
   1:  PR[91,1] = PR[90,1] + -33.551;
   1:  PR[91,2] = PR[90,2] + 9.068;
   1:L PR[91] R[100]mm/sec CNT100;
   1:  PR[91,1] = PR[90,1] + -34.430;
   1:  PR[91,2] = PR[90,2] + 7.501;
   1:L PR[91] R[100]mm/sec CNT100;
   1:  PR[91,1] = PR[90,1] + -35.135;
   1:  PR[91,2] = PR[90,2] + 5.689;
   1:L PR[91] R[100]mm/sec CNT100;
   1:  PR[91,1] = PR[90,1] + -35.593;
   1:  PR[91,2] = PR[90,2] + 4.435;
   1:L PR[91] R[100]mm/sec CNT100;
   1:  PR[91,1] = PR[90,1] + -35.968;
   1:  PR[91,2] = PR[90,2] + 2.767;
   1:L PR[91] R[100]mm/sec CNT100;
   1:  PR[91,1] = PR[90,1] + -36.105;
   1:  PR[91,2] = PR[90,2] + 0.785;
   1:L PR[91] R[100]mm/sec CNT100;
   1:  PR[91,1] = PR[90,1] + -36.251;
   1:  PR[91,2] = PR[90,2] + -0.479;
   1:L PR[91] R[100]mm/sec CNT100;
   1:  PR[91,1] = PR[90,1] + -36.125;
   1:  PR[91,2] = PR[90,2] + -2.308;
   1:L PR[91] R[100]mm/sec CNT100;
   1:  PR[91,1] = PR[90,1] + -35.980;
   1:  PR[91,2] = PR[90,2] + -3.560;
   1:L PR[91] R[100]mm/sec CNT100;
   1:  PR[91,1] = PR[90,1] + -35.599;
   1:  PR[91,2] = PR[90,2] + -5.258;
   1:L PR[91] R[100]mm/sec CNT100;
   1:  PR[91,1] = PR[90,1] + -34.901;
   1:  PR[91,2] = PR[90,2] + -7.050;
   1:L PR[91] R[100]mm/sec CNT100;
   1:  PR[91,1] = PR[90,1] + -34.418;
   1:  PR[91,2] = PR[90,2] + -8.370;
   1:L PR[91] R[100]mm/sec CNT100;
   1:  PR[91,1] = PR[90,1] + -33.551;
   1:  PR[91,2] = PR[90,2] + -9.915;
   1:L PR[91] R[100]mm/sec CNT100;
   1:  PR[91,1] = PR[90,1] + -32.666;
   1:  PR[91,2] = PR[90,2] + -11.294;
   1:L PR[91] R[100]mm/sec CNT100;
   1:  PR[91,1] = PR[90,1] + -31.670;
   1:  PR[91,2] = PR[90,2] + -12.592;
   1:L PR[91] R[100]mm/sec CNT100;
   1:  PR[91,1] = PR[90,1] + -29.115;
   1:  PR[91,2] = PR[90,2] + -15.087;
   1:L PR[91] R[100]mm/sec CNT100;
   1:  PR[91,1] = PR[90,1] + -27.990;
   1:  PR[91,2] = PR[90,2] + -15.917;
   1:L PR[91] R[100]mm/sec CNT100;
   1:  PR[91,1] = PR[90,1] + -25.960;
   1:  PR[91,2] = PR[90,2] + -17.181;
   1:L PR[91] R[100]mm/sec CNT100;
   1:  PR[91,1] = PR[90,1] + -24.821;
   1:  PR[91,2] = PR[90,2] + -17.803;
   1:L PR[91] R[100]mm/sec CNT100;
   1:  PR[91,1] = PR[90,1] + -23.734;
   1:  PR[91,2] = PR[90,2] + -18.218;
   1:L PR[91] R[100]mm/sec CNT100;
   1:  PR[91,1] = PR[90,1] + -21.040;
   1:  PR[91,2] = PR[90,2] + -19.185;
   1:L PR[91] R[100]mm/sec CNT100;
   1:  PR[91,1] = PR[90,1] + -20.183;
   1:  PR[91,2] = PR[90,2] + -19.388;
   1:L PR[91] R[100]mm/sec CNT100;
   1:  PR[91,1] = PR[90,1] + -19.265;
   1:  PR[91,2] = PR[90,2] + -19.476;
   1:L PR[91] R[100]mm/sec CNT100;
   1:  PR[91,1] = PR[90,1] + -15.999;
   1:  PR[91,2] = PR[90,2] + -19.915;
   1:L PR[91] R[100]mm/sec CNT100;
   1:  PR[91,1] = PR[90,1] + -15.397;
   1:  PR[91,2] = PR[90,2] + -19.895;
   1:L PR[91] R[100]mm/sec CNT100;
   1:  PR[91,1] = PR[90,1] + -11.643;
   1:  PR[91,2] = PR[90,2] + -19.594;
   1:L PR[91] R[100]mm/sec CNT100;
   1:  PR[91,1] = PR[90,1] + -11.254;
   1:  PR[91,2] = PR[90,2] + -19.529;
   1:L PR[91] R[100]mm/sec CNT100;
   1:  PR[91,1] = PR[90,1] + -6.938;
   1:  PR[91,2] = PR[90,2] + -18.218;
   1:L PR[91] R[100]mm/sec CNT100;
   1:  PR[91,1] = PR[90,1] + -6.827;
   1:  PR[91,2] = PR[90,2] + -18.166;
   1:L PR[91] R[100]mm/sec CNT100;
   1:  PR[91,1] = PR[90,1] + -2.906;
   1:  PR[91,2] = PR[90,2] + -15.961;
   1:L PR[91] R[100]mm/sec CNT100;
   1:  PR[91,1] = PR[90,1] + -2.454;
   1:  PR[91,2] = PR[90,2] + -15.589;
   1:L PR[91] R[100]mm/sec CNT100;
   1:  PR[91,1] = PR[90,1] + -1.862;
   1:  PR[91,2] = PR[90,2] + -15.354;
   1:L PR[91] R[100]mm/sec CNT100;
   1:  PR[91,1] = PR[90,1] + -0.836;
   1:  PR[91,2] = PR[90,2] + -14.675;
   1:L PR[91] R[100]mm/sec CNT100;
   1:  PR[91,1] = PR[90,1] + 0.716;
   1:  PR[91,2] = PR[90,2] + -15.107;
   1:L PR[91] R[100]mm/sec CNT100;
   1:  PR[91,1] = PR[90,1] + 1.350;
   1:  PR[91,2] = PR[90,2] + -15.205;
   1:L PR[91] R[100]mm/sec CNT100;
   1:  PR[91,1] = PR[90,1] + 1.836;
   1:  PR[91,2] = PR[90,2] + -15.548;
   1:L PR[91] R[100]mm/sec CNT100;
   1:  PR[91,1] = PR[90,1] + 2.083;
   1:  PR[91,2] = PR[90,2] + -15.680;
   1:L PR[91] R[100]mm/sec CNT100;
   1:  PR[91,1] = PR[90,1] + 2.413;
   1:  PR[91,2] = PR[90,2] + -15.955;
   1:L PR[91] R[100]mm/sec CNT100;
   1:  PR[91,1] = PR[90,1] + 2.424;
   1:  PR[91,2] = PR[90,2] + -15.962;
   1:L PR[91] R[100]mm/sec CNT100;
   1:  PR[91,1] = PR[90,1] + 6.341;
   1:  PR[91,2] = PR[90,2] + -18.163;
   1:L PR[91] R[100]mm/sec CNT100;
   1:  PR[91,1] = PR[90,1] + 6.452;
   1:  PR[91,2] = PR[90,2] + -18.215;
   1:L PR[91] R[100]mm/sec CNT100;
   1:  PR[91,1] = PR[90,1] + 10.771;
   1:  PR[91,2] = PR[90,2] + -19.528;
   1:L PR[91] R[100]mm/sec CNT100;
   1:  PR[91,1] = PR[90,1] + 11.160;
   1:  PR[91,2] = PR[90,2] + -19.593;
   1:L PR[91] R[100]mm/sec CNT100;
   1:  PR[91,1] = PR[90,1] + 14.914;
   1:  PR[91,2] = PR[90,2] + -19.896;
   1:L PR[91] R[100]mm/sec CNT100;
   1:  PR[91,1] = PR[90,1] + 15.555;
   1:  PR[91,2] = PR[90,2] + -19.917;
   1:L PR[91] R[100]mm/sec CNT100;
   1:  PR[91,1] = PR[90,1] + 16.328;
   1:  PR[91,2] = PR[90,2] + -19.841;
   1:L PR[91] R[100]mm/sec CNT100;
   1:  PR[91,1] = PR[90,1] + 19.648;
   1:  PR[91,2] = PR[90,2] + -19.400;
   1:L PR[91] R[100]mm/sec CNT100;
   1:  PR[91,1] = PR[90,1] + 20.528;
   1:  PR[91,2] = PR[90,2] + -19.192;
   1:L PR[91] R[100]mm/sec CNT100;
   1:  PR[91,1] = PR[90,1] + 21.660;
   1:  PR[91,2] = PR[90,2] + -18.764;
   1:L PR[91] R[100]mm/sec CNT100;
   1:  PR[91,1] = PR[90,1] + 24.353;
   1:  PR[91,2] = PR[90,2] + -17.796;
   1:L PR[91] R[100]mm/sec CNT100;
   1:  PR[91,1] = PR[90,1] + 25.467;
   1:  PR[91,2] = PR[90,2] + -17.191;
   1:L PR[91] R[100]mm/sec CNT100;
   1:  PR[91,1] = PR[90,1] + 27.497;
   1:  PR[91,2] = PR[90,2] + -15.928;
   1:L PR[91] R[100]mm/sec CNT100;
   1:  PR[91,1] = PR[90,1] + 28.608;
   1:  PR[91,2] = PR[90,2] + -15.113;
   1:L PR[91] R[100]mm/sec CNT100;
   1:  PR[91,1] = PR[90,1] + 31.161;
   1:  PR[91,2] = PR[90,2] + -12.618;
   1:L PR[91] R[100]mm/sec CNT100;
   1:  PR[91,1] = PR[90,1] + 32.169;
   1:  PR[91,2] = PR[90,2] + -11.309;
   1:L PR[91] R[100]mm/sec CNT100;
   1:  PR[91,1] = PR[90,1] + 33.057;
   1:  PR[91,2] = PR[90,2] + -9.928;
   1:L PR[91] R[100]mm/sec CNT100;
   1:  PR[91,1] = PR[90,1] + 33.945;
   1:  PR[91,2] = PR[90,2] + -8.360;
   1:L PR[91] R[100]mm/sec CNT100;
   1:  PR[91,1] = PR[90,1] + 34.644;
   1:  PR[91,2] = PR[90,2] + -6.586;
   1:L PR[91] R[100]mm/sec CNT100;
   1:  PR[91,1] = PR[90,1] + 35.102;
   1:  PR[91,2] = PR[90,2] + -5.339;
   1:L PR[91] R[100]mm/sec CNT100;
   1:  PR[91,1] = PR[90,1] + 35.480;
   1:  PR[91,2] = PR[90,2] + -3.682;
   1:L PR[91] R[100]mm/sec CNT100;
   1:  PR[91,1] = PR[90,1] + 35.626;
   1:  PR[91,2] = PR[90,2] + -1.636;
   1:L PR[91] R[100]mm/sec CNT100;
   1:  PR[91,1] = PR[90,1] + 35.771;
   1:  PR[91,2] = PR[90,2] + -0.371;
   1:L PR[91] R[100]mm/sec CNT100;
   1:  PR[91,1] = PR[90,1] + 35.636;
   1:  PR[91,2] = PR[90,2] + 1.526;
   1:L PR[91] R[100]mm/sec CNT100;
   1:  PR[91,1] = PR[90,1] + 35.491;
   1:  PR[91,2] = PR[90,2] + 2.783;
   1:L PR[91] R[100]mm/sec CNT100;
   1:  PR[91,1] = PR[90,1] + 35.109;
   1:  PR[91,2] = PR[90,2] + 4.464;
   1:L PR[91] R[100]mm/sec CNT100;
   1:  PR[91,1] = PR[90,1] + 34.414;
   1:  PR[91,2] = PR[90,2] + 6.222;
   1:L PR[91] R[100]mm/sec CNT100;
   1:  PR[91,1] = PR[90,1] + 33.931;
   1:  PR[91,2] = PR[90,2] + 7.537;
   1:L PR[91] R[100]mm/sec CNT100;
   1:  PR[91,1] = PR[90,1] + 33.057;
   1:  PR[91,2] = PR[90,2] + 9.081;
   1:L PR[91] R[100]mm/sec CNT100;
   1:  PR[91,1] = PR[90,1] + 32.169;
   1:  PR[91,2] = PR[90,2] + 10.462;
   1:L PR[91] R[100]mm/sec CNT100;
   1:  PR[91,1] = PR[90,1] + 31.161;
   1:  PR[91,2] = PR[90,2] + 11.771;
   1:L PR[91] R[100]mm/sec CNT100;
   1:  PR[91,1] = PR[90,1] + 28.608;
   1:  PR[91,2] = PR[90,2] + 14.265;
   1:L PR[91] R[100]mm/sec CNT100;
   1:  PR[91,1] = PR[90,1] + 27.497;
   1:  PR[91,2] = PR[90,2] + 15.081;
   1:L PR[91] R[100]mm/sec CNT100;
   1:  PR[91,1] = PR[90,1] + 25.467;
   1:  PR[91,2] = PR[90,2] + 16.344;
   1:L PR[91] R[100]mm/sec CNT100;
   1:  PR[91,1] = PR[90,1] + 24.334;
   1:  PR[91,2] = PR[90,2] + 16.959;
   1:L PR[91] R[100]mm/sec CNT100;
   1:  PR[91,1] = PR[90,1] + 23.243;
   1:  PR[91,2] = PR[90,2] + 17.373;
   1:L PR[91] R[100]mm/sec CNT100;
   1:  PR[91,1] = PR[90,1] + 20.547;
   1:  PR[91,2] = PR[90,2] + 18.340;
   1:L PR[91] R[100]mm/sec CNT100;
   1:  PR[91,1] = PR[90,1] + 19.693;
   1:  PR[91,2] = PR[90,2] + 18.542;
   1:L PR[91] R[100]mm/sec CNT100;
   1:  PR[91,1] = PR[90,1] + 18.779;
   1:  PR[91,2] = PR[90,2] + 18.628;
   1:L PR[91] R[100]mm/sec CNT100;
   1:  PR[91,1] = PR[90,1] + 15.512;
   1:  PR[91,2] = PR[90,2] + 19.069;
   1:L PR[91] R[100]mm/sec CNT100;
   1:  PR[91,1] = PR[90,1] + 14.914;
   1:  PR[91,2] = PR[90,2] + 19.048;
   1:L PR[91] R[100]mm/sec CNT100;
   1:  PR[91,1] = PR[90,1] + 11.160;
   1:  PR[91,2] = PR[90,2] + 18.746;
   1:L PR[91] R[100]mm/sec CNT100;
   1:  PR[91,1] = PR[90,1] + 10.771;
   1:  PR[91,2] = PR[90,2] + 18.681;
   1:L PR[91] R[100]mm/sec CNT100;
   1:  PR[91,1] = PR[90,1] + 6.452;
   1:  PR[91,2] = PR[90,2] + 17.368;
   1:L PR[91] R[100]mm/sec CNT100;
   1:  PR[91,1] = PR[90,1] + 6.342;
   1:  PR[91,2] = PR[90,2] + 17.316;
   1:L PR[91] R[100]mm/sec CNT100;
   1:  PR[91,1] = PR[90,1] + 2.424;
   1:  PR[91,2] = PR[90,2] + 15.115;
   1:L PR[91] R[100]mm/sec CNT100;
   1:  PR[91,1] = PR[90,1] + 2.082;
   1:  PR[91,2] = PR[90,2] + 14.833;
   1:L PR[91] R[100]mm/sec CNT100;
   1:  PR[91,1] = PR[90,1] + 1.831;
   1:  PR[91,2] = PR[90,2] + 14.697;
   1:L PR[91] R[100]mm/sec CNT100;
   1:  PR[91,1] = PR[90,1] + 1.354;
   1:  PR[91,2] = PR[90,2] + 14.357;
   1:L PR[91] R[100]mm/sec CNT100;
   1:  PR[91,1] = PR[90,1] + 0.863;
   1:  PR[91,2] = PR[90,2] + 14.282;
   1:L PR[91] R[100]mm/sec CNT100;
   1:  PR[91,1] = PR[90,1] + 0.271;
   1:  PR[91,2] = PR[90,2] + 14.034;
   1:L PR[91] R[100]mm/sec CNT100;
   1:  PR[91] = PR[90];
   1:  PR[91,1] = PR[90,1] + -0.906;
   1:  PR[91,2] = PR[90,2] + 14.621;
   1:  PR[91,3] = PR[90,3] + 36.595;
   1:L PR[91] R[100]mm/sec CNT100;
   1:  PR[91,1] = PR[90,1] + -1.737;
   1:  PR[91,2] = PR[90,2] + 15.006;
   1:L PR[91] R[100]mm/sec CNT100;
   1:  PR[91,1] = PR[90,1] + -2.132;
   1:  PR[91,2] = PR[90,2] + 15.132;
   1:L PR[91] R[100]mm/sec CNT100;
   1:  PR[91,1] = PR[90,1] + -6.402;
   1:  PR[91,2] = PR[90,2] + 17.485;
   1:L PR[91] R[100]mm/sec CNT100;
   1:  PR[91,1] = PR[90,1] + -10.845;
   1:  PR[91,2] = PR[90,2] + 18.832;
   1:L PR[91] R[100]mm/sec CNT100;
   1:  PR[91,1] = PR[90,1] + -10.901;
   1:  PR[91,2] = PR[90,2] + 18.841;
   1:L PR[91] R[100]mm/sec CNT100;
   1:  PR[91,1] = PR[90,1] + -15.199;
   1:  PR[91,2] = PR[90,2] + 19.185;
   1:L PR[91] R[100]mm/sec CNT100;
   1:  PR[91,1] = PR[90,1] + -15.522;
   1:  PR[91,2] = PR[90,2] + 19.196;
   1:L PR[91] R[100]mm/sec CNT100;
   1:  PR[91,1] = PR[90,1] + -15.935;
   1:  PR[91,2] = PR[90,2] + 19.155;
   1:L PR[91] R[100]mm/sec CNT100;
   1:  PR[91,1] = PR[90,1] + -19.834;
   1:  PR[91,2] = PR[90,2] + 18.637;
   1:L PR[91] R[100]mm/sec CNT100;
   1:  PR[91,1] = PR[90,1] + -20.377;
   1:  PR[91,2] = PR[90,2] + 18.508;
   1:L PR[91] R[100]mm/sec CNT100;
   1:  PR[91,1] = PR[90,1] + -21.139;
   1:  PR[91,2] = PR[90,2] + 18.219;
   1:L PR[91] R[100]mm/sec CNT100;
   1:  PR[91,1] = PR[90,1] + -24.417;
   1:  PR[91,2] = PR[90,2] + 17.039;
   1:L PR[91] R[100]mm/sec CNT100;
   1:  PR[91,1] = PR[90,1] + -25.209;
   1:  PR[91,2] = PR[90,2] + 16.607;
   1:L PR[91] R[100]mm/sec CNT100;
   1:  PR[91,1] = PR[90,1] + -27.740;
   1:  PR[91,2] = PR[90,2] + 15.030;
   1:L PR[91] R[100]mm/sec CNT100;
   1:  PR[91,1] = PR[90,1] + -28.583;
   1:  PR[91,2] = PR[90,2] + 14.408;
   1:L PR[91] R[100]mm/sec CNT100;
   1:  PR[91,1] = PR[90,1] + -31.305;
   1:  PR[91,2] = PR[90,2] + 11.747;
   1:L PR[91] R[100]mm/sec CNT100;
   1:  PR[91,1] = PR[90,1] + -32.081;
   1:  PR[91,2] = PR[90,2] + 10.737;
   1:L PR[91] R[100]mm/sec CNT100;
   1:  PR[91,1] = PR[90,1] + -33.285;
   1:  PR[91,2] = PR[90,2] + 8.860;
   1:L PR[91] R[100]mm/sec CNT100;
   1:  PR[91,1] = PR[90,1] + -33.988;
   1:  PR[91,2] = PR[90,2] + 7.608;
   1:L PR[91] R[100]mm/sec CNT100;
   1:  PR[91,1] = PR[90,1] + -34.555;
   1:  PR[91,2] = PR[90,2] + 6.149;
   1:L PR[91] R[100]mm/sec CNT100;
   1:  PR[91,1] = PR[90,1] + -35.218;
   1:  PR[91,2] = PR[90,2] + 4.337;
   1:L PR[91] R[100]mm/sec CNT100;
   1:  PR[91,1] = PR[90,1] + -35.516;
   1:  PR[91,2] = PR[90,2] + 3.007;
   1:L PR[91] R[100]mm/sec CNT100;
   1:  PR[91,1] = PR[90,1] + -35.629;
   1:  PR[91,2] = PR[90,2] + 1.384;
   1:L PR[91] R[100]mm/sec CNT100;
   1:  PR[91,1] = PR[90,1] + -35.844;
   1:  PR[91,2] = PR[90,2] + -0.479;
   1:L PR[91] R[100]mm/sec CNT100;
   1:  PR[91,1] = PR[90,1] + -35.742;
   1:  PR[91,2] = PR[90,2] + -1.958;
   1:L PR[91] R[100]mm/sec CNT100;
   1:  PR[91,1] = PR[90,1] + -35.528;
   1:  PR[91,2] = PR[90,2] + -3.801;
   1:L PR[91] R[100]mm/sec CNT100;
   1:  PR[91,1] = PR[90,1] + -35.224;
   1:  PR[91,2] = PR[90,2] + -5.160;
   1:L PR[91] R[100]mm/sec CNT100;
   1:  PR[91,1] = PR[90,1] + -34.654;
   1:  PR[91,2] = PR[90,2] + -6.622;
   1:L PR[91] R[100]mm/sec CNT100;
   1:  PR[91,1] = PR[90,1] + -33.976;
   1:  PR[91,2] = PR[90,2] + -8.476;
   1:L PR[91] R[100]mm/sec CNT100;
   1:  PR[91,1] = PR[90,1] + -33.285;
   1:  PR[91,2] = PR[90,2] + -9.707;
   1:L PR[91] R[100]mm/sec CNT100;
   1:  PR[91,1] = PR[90,1] + -32.081;
   1:  PR[91,2] = PR[90,2] + -11.584;
   1:L PR[91] R[100]mm/sec CNT100;
   1:  PR[91,1] = PR[90,1] + -31.305;
   1:  PR[91,2] = PR[90,2] + -12.594;
   1:L PR[91] R[100]mm/sec CNT100;
   1:  PR[91,1] = PR[90,1] + -28.583;
   1:  PR[91,2] = PR[90,2] + -15.255;
   1:L PR[91] R[100]mm/sec CNT100;
   1:  PR[91,1] = PR[90,1] + -27.740;
   1:  PR[91,2] = PR[90,2] + -15.877;
   1:L PR[91] R[100]mm/sec CNT100;
   1:  PR[91,1] = PR[90,1] + -25.208;
   1:  PR[91,2] = PR[90,2] + -17.454;
   1:L PR[91] R[100]mm/sec CNT100;
   1:  PR[91,1] = PR[90,1] + -24.396;
   1:  PR[91,2] = PR[90,2] + -17.898;
   1:L PR[91] R[100]mm/sec CNT100;
   1:  PR[91,1] = PR[90,1] + -23.616;
   1:  PR[91,2] = PR[90,2] + -18.195;
   1:L PR[91] R[100]mm/sec CNT100;
   1:  PR[91,1] = PR[90,1] + -20.398;
   1:  PR[91,2] = PR[90,2] + -19.351;
   1:L PR[91] R[100]mm/sec CNT100;
   1:  PR[91,1] = PR[90,1] + -19.877;
   1:  PR[91,2] = PR[90,2] + -19.474;
   1:L PR[91] R[100]mm/sec CNT100;
   1:  PR[91,1] = PR[90,1] + -19.263;
   1:  PR[91,2] = PR[90,2] + -19.533;
   1:L PR[91] R[100]mm/sec CNT100;
   1:  PR[91,1] = PR[90,1] + -15.479;
   1:  PR[91,2] = PR[90,2] + -20.042;
   1:L PR[91] R[100]mm/sec CNT100;
   1:  PR[91,1] = PR[90,1] + -15.199;
   1:  PR[91,2] = PR[90,2] + -20.033;
   1:L PR[91] R[100]mm/sec CNT100;
   1:  PR[91,1] = PR[90,1] + -10.901;
   1:  PR[91,2] = PR[90,2] + -19.688;
   1:L PR[91] R[100]mm/sec CNT100;
   1:  PR[91,1] = PR[90,1] + -10.845;
   1:  PR[91,2] = PR[90,2] + -19.679;
   1:L PR[91] R[100]mm/sec CNT100;
   1:  PR[91,1] = PR[90,1] + -6.401;
   1:  PR[91,2] = PR[90,2] + -18.332;
   1:L PR[91] R[100]mm/sec CNT100;
   1:  PR[91,1] = PR[90,1] + -2.136;
   1:  PR[91,2] = PR[90,2] + -15.981;
   1:L PR[91] R[100]mm/sec CNT100;
   1:  PR[91,1] = PR[90,1] + -1.638;
   1:  PR[91,2] = PR[90,2] + -15.821;
   1:L PR[91] R[100]mm/sec CNT100;
   1:  PR[91,1] = PR[90,1] + -1.622;
   1:  PR[91,2] = PR[90,2] + -15.815;
   1:L PR[91] R[100]mm/sec CNT100;
   1:  PR[91,1] = PR[90,1] + -0.788;
   1:  PR[91,2] = PR[90,2] + -15.263;
   1:L PR[91] R[100]mm/sec CNT100;
   1:  PR[91,1] = PR[90,1] + 0.384;
   1:  PR[91,2] = PR[90,2] + -15.590;
   1:L PR[91] R[100]mm/sec CNT100;
   1:  PR[91,1] = PR[90,1] + 1.398;
   1:  PR[91,2] = PR[90,2] + -15.747;
   1:L PR[91] R[100]mm/sec CNT100;
   1:  PR[91,1] = PR[90,1] + 1.978;
   1:  PR[91,2] = PR[90,2] + -16.161;
   1:L PR[91] R[100]mm/sec CNT100;
   1:  PR[91,1] = PR[90,1] + 5.916;
   1:  PR[91,2] = PR[90,2] + -18.330;
   1:L PR[91] R[100]mm/sec CNT100;
   1:  PR[91,1] = PR[90,1] + 10.362;
   1:  PR[91,2] = PR[90,2] + -19.678;
   1:L PR[91] R[100]mm/sec CNT100;
   1:  PR[91,1] = PR[90,1] + 10.418;
   1:  PR[91,2] = PR[90,2] + -19.687;
   1:L PR[91] R[100]mm/sec CNT100;
   1:  PR[91,1] = PR[90,1] + 14.716;
   1:  PR[91,2] = PR[90,2] + -20.033;
   1:L PR[91] R[100]mm/sec CNT100;
   1:  PR[91,1] = PR[90,1] + 15.037;
   1:  PR[91,2] = PR[90,2] + -20.044;
   1:L PR[91] R[100]mm/sec CNT100;
   1:  PR[91,1] = PR[90,1] + 15.446;
   1:  PR[91,2] = PR[90,2] + -20.004;
   1:L PR[91] R[100]mm/sec CNT100;
   1:  PR[91,1] = PR[90,1] + 19.345;
   1:  PR[91,2] = PR[90,2] + -19.485;
   1:L PR[91] R[100]mm/sec CNT100;
   1:  PR[91,1] = PR[90,1] + 19.888;
   1:  PR[91,2] = PR[90,2] + -19.357;
   1:L PR[91] R[100]mm/sec CNT100;
   1:  PR[91,1] = PR[90,1] + 20.651;
   1:  PR[91,2] = PR[90,2] + -19.069;
   1:L PR[91] R[100]mm/sec CNT100;
   1:  PR[91,1] = PR[90,1] + 23.931;
   1:  PR[91,2] = PR[90,2] + -17.890;
   1:L PR[91] R[100]mm/sec CNT100;
   1:  PR[91,1] = PR[90,1] + 24.719;
   1:  PR[91,2] = PR[90,2] + -17.462;
   1:L PR[91] R[100]mm/sec CNT100;
   1:  PR[91,1] = PR[90,1] + 27.251;
   1:  PR[91,2] = PR[90,2] + -15.887;
   1:L PR[91] R[100]mm/sec CNT100;
   1:  PR[91,1] = PR[90,1] + 28.082;
   1:  PR[91,2] = PR[90,2] + -15.277;
   1:L PR[91] R[100]mm/sec CNT100;
   1:  PR[91,1] = PR[90,1] + 30.802;
   1:  PR[91,2] = PR[90,2] + -12.615;
   1:L PR[91] R[100]mm/sec CNT100;
   1:  PR[91,1] = PR[90,1] + 31.587;
   1:  PR[91,2] = PR[90,2] + -11.595;
   1:L PR[91] R[100]mm/sec CNT100;
   1:  PR[91,1] = PR[90,1] + 32.794;
   1:  PR[91,2] = PR[90,2] + -9.717;
   1:L PR[91] R[100]mm/sec CNT100;
   1:  PR[91,1] = PR[90,1] + 33.504;
   1:  PR[91,2] = PR[90,2] + -8.463;
   1:L PR[91] R[100]mm/sec CNT100;
   1:  PR[91,1] = PR[90,1] + 34.067;
   1:  PR[91,2] = PR[90,2] + -7.036;
   1:L PR[91] R[100]mm/sec CNT100;
   1:  PR[91,1] = PR[90,1] + 34.729;
   1:  PR[91,2] = PR[90,2] + -5.233;
   1:L PR[91] R[100]mm/sec CNT100;
   1:  PR[91,1] = PR[90,1] + 35.030;
   1:  PR[91,2] = PR[90,2] + -3.913;
   1:L PR[91] R[100]mm/sec CNT100;
   1:  PR[91,1] = PR[90,1] + 35.150;
   1:  PR[91,2] = PR[90,2] + -2.237;
   1:L PR[91] R[100]mm/sec CNT100;
   1:  PR[91,1] = PR[90,1] + 35.364;
   1:  PR[91,2] = PR[90,2] + -0.371;
   1:L PR[91] R[100]mm/sec CNT100;
   1:  PR[91,1] = PR[90,1] + 35.255;
   1:  PR[91,2] = PR[90,2] + 1.165;
   1:L PR[91] R[100]mm/sec CNT100;
   1:  PR[91,1] = PR[90,1] + 35.042;
   1:  PR[91,2] = PR[90,2] + 3.015;
   1:L PR[91] R[100]mm/sec CNT100;
   1:  PR[91,1] = PR[90,1] + 34.736;
   1:  PR[91,2] = PR[90,2] + 4.358;
   1:L PR[91] R[100]mm/sec CNT100;
   1:  PR[91,1] = PR[90,1] + 34.169;
   1:  PR[91,2] = PR[90,2] + 5.793;
   1:L PR[91] R[100]mm/sec CNT100;
   1:  PR[91,1] = PR[90,1] + 33.490;
   1:  PR[91,2] = PR[90,2] + 7.640;
   1:L PR[91] R[100]mm/sec CNT100;
   1:  PR[91,1] = PR[90,1] + 32.794;
   1:  PR[91,2] = PR[90,2] + 8.870;
   1:L PR[91] R[100]mm/sec CNT100;
   1:  PR[91,1] = PR[90,1] + 31.587;
   1:  PR[91,2] = PR[90,2] + 10.747;
   1:L PR[91] R[100]mm/sec CNT100;
   1:  PR[91,1] = PR[90,1] + 30.802;
   1:  PR[91,2] = PR[90,2] + 11.767;
   1:L PR[91] R[100]mm/sec CNT100;
   1:  PR[91,1] = PR[90,1] + 28.082;
   1:  PR[91,2] = PR[90,2] + 14.429;
   1:L PR[91] R[100]mm/sec CNT100;
   1:  PR[91,1] = PR[90,1] + 27.251;
   1:  PR[91,2] = PR[90,2] + 15.039;
   1:L PR[91] R[100]mm/sec CNT100;
   1:  PR[91,1] = PR[90,1] + 24.719;
   1:  PR[91,2] = PR[90,2] + 16.614;
   1:L PR[91] R[100]mm/sec CNT100;
   1:  PR[91,1] = PR[90,1] + 23.912;
   1:  PR[91,2] = PR[90,2] + 17.052;
   1:L PR[91] R[100]mm/sec CNT100;
   1:  PR[91,1] = PR[90,1] + 23.128;
   1:  PR[91,2] = PR[90,2] + 17.350;
   1:L PR[91] R[100]mm/sec CNT100;
   1:  PR[91,1] = PR[90,1] + 19.908;
   1:  PR[91,2] = PR[90,2] + 18.505;
   1:L PR[91] R[100]mm/sec CNT100;
   1:  PR[91,1] = PR[90,1] + 19.390;
   1:  PR[91,2] = PR[90,2] + 18.628;
   1:L PR[91] R[100]mm/sec CNT100;
   1:  PR[91,1] = PR[90,1] + 18.778;
   1:  PR[91,2] = PR[90,2] + 18.685;
   1:L PR[91] R[100]mm/sec CNT100;
   1:  PR[91,1] = PR[90,1] + 14.994;
   1:  PR[91,2] = PR[90,2] + 19.195;
   1:L PR[91] R[100]mm/sec CNT100;
   1:  PR[91,1] = PR[90,1] + 14.716;
   1:  PR[91,2] = PR[90,2] + 19.186;
   1:L PR[91] R[100]mm/sec CNT100;
   1:  PR[91,1] = PR[90,1] + 10.418;
   1:  PR[91,2] = PR[90,2] + 18.840;
   1:L PR[91] R[100]mm/sec CNT100;
   1:  PR[91,1] = PR[90,1] + 10.362;
   1:  PR[91,2] = PR[90,2] + 18.830;
   1:L PR[91] R[100]mm/sec CNT100;
   1:  PR[91,1] = PR[90,1] + 5.916;
   1:  PR[91,2] = PR[90,2] + 17.483;
   1:L PR[91] R[100]mm/sec CNT100;
   1:  PR[91,1] = PR[90,1] + 1.978;
   1:  PR[91,2] = PR[90,2] + 15.314;
   1:L PR[91] R[100]mm/sec CNT100;
   1:  PR[91,1] = PR[90,1] + 1.394;
   1:  PR[91,2] = PR[90,2] + 14.896;
   1:L PR[91] R[100]mm/sec CNT100;
   1:  PR[91,1] = PR[90,1] + 0.531;
   1:  PR[91,2] = PR[90,2] + 14.765;
   1:L PR[91] R[100]mm/sec CNT100;
   1:  PR[91,1] = PR[90,1] + 0.191;
   1:  PR[91,2] = PR[90,2] + 14.622;
   1:L PR[91] R[100]mm/sec CNT100;
   1:  PR[91] = PR[90];
   1:  PR[91,1] = PR[90,1] + -2.097;
   1:  PR[91,2] = PR[90,2] + 15.618;
   1:  PR[91,3] = PR[90,3] + 37.895;
   1:L PR[91] R[100]mm/sec CNT100;
   1:  PR[91,1] = PR[90,1] + -5.253;
   1:  PR[91,2] = PR[90,2] + 17.345;
   1:L PR[91] R[100]mm/sec CNT100;
   1:  PR[91,1] = PR[90,1] + -5.848;
   1:  PR[91,2] = PR[90,2] + 17.646;
   1:L PR[91] R[100]mm/sec CNT100;
   1:  PR[91,1] = PR[90,1] + -10.319;
   1:  PR[91,2] = PR[90,2] + 18.953;
   1:L PR[91] R[100]mm/sec CNT100;
   1:  PR[91,1] = PR[90,1] + -15.016;
   1:  PR[91,2] = PR[90,2] + 19.315;
   1:L PR[91] R[100]mm/sec CNT100;
   1:  PR[91,1] = PR[90,1] + -19.530;
   1:  PR[91,2] = PR[90,2] + 18.722;
   1:L PR[91] R[100]mm/sec CNT100;
   1:  PR[91,1] = PR[90,1] + -19.752;
   1:  PR[91,2] = PR[90,2] + 18.670;
   1:L PR[91] R[100]mm/sec CNT100;
   1:  PR[91,1] = PR[90,1] + -23.990;
   1:  PR[91,2] = PR[90,2] + 17.135;
   1:L PR[91] R[100]mm/sec CNT100;
   1:  PR[91,1] = PR[90,1] + -24.457;
   1:  PR[91,2] = PR[90,2] + 16.880;
   1:L PR[91] R[100]mm/sec CNT100;
   1:  PR[91,1] = PR[90,1] + -27.491;
   1:  PR[91,2] = PR[90,2] + 14.990;
   1:L PR[91] R[100]mm/sec CNT100;
   1:  PR[91,1] = PR[90,1] + -28.052;
   1:  PR[91,2] = PR[90,2] + 14.576;
   1:L PR[91] R[100]mm/sec CNT100;
   1:  PR[91,1] = PR[90,1] + -30.941;
   1:  PR[91,2] = PR[90,2] + 11.749;
   1:L PR[91] R[100]mm/sec CNT100;
   1:  PR[91,1] = PR[90,1] + -31.495;
   1:  PR[91,2] = PR[90,2] + 11.027;
   1:L PR[91] R[100]mm/sec CNT100;
   1:  PR[91,1] = PR[90,1] + -33.019;
   1:  PR[91,2] = PR[90,2] + 8.652;
   1:L PR[91] R[100]mm/sec CNT100;
   1:  PR[91,1] = PR[90,1] + -33.545;
   1:  PR[91,2] = PR[90,2] + 7.714;
   1:L PR[91] R[100]mm/sec CNT100;
   1:  PR[91,1] = PR[90,1] + -33.976;
   1:  PR[91,2] = PR[90,2] + 6.608;
   1:L PR[91] R[100]mm/sec CNT100;
   1:  PR[91,1] = PR[90,1] + -34.843;
   1:  PR[91,2] = PR[90,2] + 4.238;
   1:L PR[91] R[100]mm/sec CNT100;
   1:  PR[91,1] = PR[90,1] + -35.065;
   1:  PR[91,2] = PR[90,2] + 3.248;
   1:L PR[91] R[100]mm/sec CNT100;
   1:  PR[91,1] = PR[90,1] + -35.153;
   1:  PR[91,2] = PR[90,2] + 1.982;
   1:L PR[91] R[100]mm/sec CNT100;
   1:  PR[91,1] = PR[90,1] + -35.437;
   1:  PR[91,2] = PR[90,2] + -0.479;
   1:L PR[91] R[100]mm/sec CNT100;
   1:  PR[91,1] = PR[90,1] + -35.359;
   1:  PR[91,2] = PR[90,2] + -1.608;
   1:L PR[91] R[100]mm/sec CNT100;
   1:  PR[91,1] = PR[90,1] + -35.077;
   1:  PR[91,2] = PR[90,2] + -4.042;
   1:L PR[91] R[100]mm/sec CNT100;
   1:  PR[91,1] = PR[90,1] + -34.849;
   1:  PR[91,2] = PR[90,2] + -5.061;
   1:L PR[91] R[100]mm/sec CNT100;
   1:  PR[91,1] = PR[90,1] + -34.407;
   1:  PR[91,2] = PR[90,2] + -6.195;
   1:L PR[91] R[100]mm/sec CNT100;
   1:  PR[91,1] = PR[90,1] + -33.533;
   1:  PR[91,2] = PR[90,2] + -8.583;
   1:L PR[91] R[100]mm/sec CNT100;
   1:  PR[91,1] = PR[90,1] + -33.019;
   1:  PR[91,2] = PR[90,2] + -9.499;
   1:L PR[91] R[100]mm/sec CNT100;
   1:  PR[91,1] = PR[90,1] + -31.495;
   1:  PR[91,2] = PR[90,2] + -11.874;
   1:L PR[91] R[100]mm/sec CNT100;
   1:  PR[91,1] = PR[90,1] + -30.941;
   1:  PR[91,2] = PR[90,2] + -12.597;
   1:L PR[91] R[100]mm/sec CNT100;
   1:  PR[91,1] = PR[90,1] + -28.051;
   1:  PR[91,2] = PR[90,2] + -15.424;
   1:L PR[91] R[100]mm/sec CNT100;
   1:  PR[91,1] = PR[90,1] + -27.491;
   1:  PR[91,2] = PR[90,2] + -15.837;
   1:L PR[91] R[100]mm/sec CNT100;
   1:  PR[91,1] = PR[90,1] + -24.457;
   1:  PR[91,2] = PR[90,2] + -17.727;
   1:L PR[91] R[100]mm/sec CNT100;
   1:  PR[91,1] = PR[90,1] + -23.971;
   1:  PR[91,2] = PR[90,2] + -17.992;
   1:L PR[91] R[100]mm/sec CNT100;
   1:  PR[91,1] = PR[90,1] + -23.498;
   1:  PR[91,2] = PR[90,2] + -18.173;
   1:L PR[91] R[100]mm/sec CNT100;
   1:  PR[91,1] = PR[90,1] + -19.755;
   1:  PR[91,2] = PR[90,2] + -19.516;
   1:L PR[91] R[100]mm/sec CNT100;
   1:  PR[91,1] = PR[90,1] + -19.571;
   1:  PR[91,2] = PR[90,2] + -19.560;
   1:L PR[91] R[100]mm/sec CNT100;
   1:  PR[91,1] = PR[90,1] + -19.261;
   1:  PR[91,2] = PR[90,2] + -19.590;
   1:L PR[91] R[100]mm/sec CNT100;
   1:  PR[91,1] = PR[90,1] + -15.011;
   1:  PR[91,2] = PR[90,2] + -20.162;
   1:L PR[91] R[100]mm/sec CNT100;
   1:  PR[91,1] = PR[90,1] + -10.319;
   1:  PR[91,2] = PR[90,2] + -19.800;
   1:L PR[91] R[100]mm/sec CNT100;
   1:  PR[91,1] = PR[90,1] + -5.848;
   1:  PR[91,2] = PR[90,2] + -18.493;
   1:L PR[91] R[100]mm/sec CNT100;
   1:  PR[91,1] = PR[90,1] + -5.233;
   1:  PR[91,2] = PR[90,2] + -18.182;
   1:L PR[91] R[100]mm/sec CNT100;
   1:  PR[91,1] = PR[90,1] + -2.098;
   1:  PR[91,2] = PR[90,2] + -16.466;
   1:L PR[91] R[100]mm/sec CNT100;
   1:  PR[91,1] = PR[90,1] + -0.302;
   1:  PR[91,2] = PR[90,2] + -15.887;
   1:L PR[91] R[100]mm/sec CNT100;
   1:  PR[91,1] = PR[90,1] + 0.369;
   1:  PR[91,2] = PR[90,2] + -16.121;
   1:L PR[91] R[100]mm/sec CNT100;
   1:  PR[91,1] = PR[90,1] + 1.439;
   1:  PR[91,2] = PR[90,2] + -16.285;
   1:L PR[91] R[100]mm/sec CNT100;
   1:  PR[91,1] = PR[90,1] + 1.941;
   1:  PR[91,2] = PR[90,2] + -16.645;
   1:L PR[91] R[100]mm/sec CNT100;
   1:  PR[91,1] = PR[90,1] + 4.765;
   1:  PR[91,2] = PR[90,2] + -18.189;
   1:L PR[91] R[100]mm/sec CNT100;
   1:  PR[91,1] = PR[90,1] + 5.363;
   1:  PR[91,2] = PR[90,2] + -18.491;
   1:L PR[91] R[100]mm/sec CNT100;
   1:  PR[91,1] = PR[90,1] + 9.835;
   1:  PR[91,2] = PR[90,2] + -19.798;
   1:L PR[91] R[100]mm/sec CNT100;
   1:  PR[91,1] = PR[90,1] + 14.531;
   1:  PR[91,2] = PR[90,2] + -20.162;
   1:L PR[91] R[100]mm/sec CNT100;
   1:  PR[91,1] = PR[90,1] + 19.044;
   1:  PR[91,2] = PR[90,2] + -19.570;
   1:L PR[91] R[100]mm/sec CNT100;
   1:  PR[91,1] = PR[90,1] + 19.265;
   1:  PR[91,2] = PR[90,2] + -19.518;
   1:L PR[91] R[100]mm/sec CNT100;
   1:  PR[91,1] = PR[90,1] + 23.506;
   1:  PR[91,2] = PR[90,2] + -17.984;
   1:L PR[91] R[100]mm/sec CNT100;
   1:  PR[91,1] = PR[90,1] + 23.971;
   1:  PR[91,2] = PR[90,2] + -17.732;
   1:L PR[91] R[100]mm/sec CNT100;
   1:  PR[91,1] = PR[90,1] + 27.004;
   1:  PR[91,2] = PR[90,2] + -15.845;
   1:L PR[91] R[100]mm/sec CNT100;
   1:  PR[91,1] = PR[90,1] + 27.556;
   1:  PR[91,2] = PR[90,2] + -15.440;
   1:L PR[91] R[100]mm/sec CNT100;
   1:  PR[91,1] = PR[90,1] + 30.443;
   1:  PR[91,2] = PR[90,2] + -12.611;
   1:L PR[91] R[100]mm/sec CNT100;
   1:  PR[91,1] = PR[90,1] + 31.005;
   1:  PR[91,2] = PR[90,2] + -11.881;
   1:L PR[91] R[100]mm/sec CNT100;
   1:  PR[91,1] = PR[90,1] + 32.531;
   1:  PR[91,2] = PR[90,2] + -9.506;
   1:L PR[91] R[100]mm/sec CNT100;
   1:  PR[91,1] = PR[90,1] + 33.064;
   1:  PR[91,2] = PR[90,2] + -8.566;
   1:L PR[91] R[100]mm/sec CNT100;
   1:  PR[91,1] = PR[90,1] + 33.490;
   1:  PR[91,2] = PR[90,2] + -7.485;
   1:L PR[91] R[100]mm/sec CNT100;
   1:  PR[91,1] = PR[90,1] + 34.356;
   1:  PR[91,2] = PR[90,2] + -5.127;
   1:L PR[91] R[100]mm/sec CNT100;
   1:  PR[91,1] = PR[90,1] + 34.580;
   1:  PR[91,2] = PR[90,2] + -4.145;
   1:L PR[91] R[100]mm/sec CNT100;
   1:  PR[91,1] = PR[90,1] + 34.673;
   1:  PR[91,2] = PR[90,2] + -2.838;
   1:L PR[91] R[100]mm/sec CNT100;
   1:  PR[91,1] = PR[90,1] + 34.957;
   1:  PR[91,2] = PR[90,2] + -0.371;
   1:L PR[91] R[100]mm/sec CNT100;
   1:  PR[91,1] = PR[90,1] + 34.874;
   1:  PR[91,2] = PR[90,2] + 0.804;
   1:L PR[91] R[100]mm/sec CNT100;
   1:  PR[91,1] = PR[90,1] + 34.592;
   1:  PR[91,2] = PR[90,2] + 3.246;
   1:L PR[91] R[100]mm/sec CNT100;
   1:  PR[91,1] = PR[90,1] + 34.363;
   1:  PR[91,2] = PR[90,2] + 4.252;
   1:L PR[91] R[100]mm/sec CNT100;
   1:  PR[91,1] = PR[90,1] + 33.923;
   1:  PR[91,2] = PR[90,2] + 5.364;
   1:L PR[91] R[100]mm/sec CNT100;
   1:  PR[91,1] = PR[90,1] + 33.050;
   1:  PR[91,2] = PR[90,2] + 7.743;
   1:L PR[91] R[100]mm/sec CNT100;
   1:  PR[91,1] = PR[90,1] + 32.531;
   1:  PR[91,2] = PR[90,2] + 8.659;
   1:L PR[91] R[100]mm/sec CNT100;
   1:  PR[91,1] = PR[90,1] + 31.005;
   1:  PR[91,2] = PR[90,2] + 11.033;
   1:L PR[91] R[100]mm/sec CNT100;
   1:  PR[91,1] = PR[90,1] + 30.443;
   1:  PR[91,2] = PR[90,2] + 11.764;
   1:L PR[91] R[100]mm/sec CNT100;
   1:  PR[91,1] = PR[90,1] + 27.556;
   1:  PR[91,2] = PR[90,2] + 14.593;
   1:L PR[91] R[100]mm/sec CNT100;
   1:  PR[91,1] = PR[90,1] + 27.004;
   1:  PR[91,2] = PR[90,2] + 14.998;
   1:L PR[91] R[100]mm/sec CNT100;
   1:  PR[91,1] = PR[90,1] + 23.971;
   1:  PR[91,2] = PR[90,2] + 16.885;
   1:L PR[91] R[100]mm/sec CNT100;
   1:  PR[91,1] = PR[90,1] + 23.489;
   1:  PR[91,2] = PR[90,2] + 17.146;
   1:L PR[91] R[100]mm/sec CNT100;
   1:  PR[91,1] = PR[90,1] + 23.013;
   1:  PR[91,2] = PR[90,2] + 17.327;
   1:L PR[91] R[100]mm/sec CNT100;
   1:  PR[91,1] = PR[90,1] + 19.268;
   1:  PR[91,2] = PR[90,2] + 18.670;
   1:L PR[91] R[100]mm/sec CNT100;
   1:  PR[91,1] = PR[90,1] + 19.087;
   1:  PR[91,2] = PR[90,2] + 18.713;
   1:L PR[91] R[100]mm/sec CNT100;
   1:  PR[91,1] = PR[90,1] + 18.778;
   1:  PR[91,2] = PR[90,2] + 18.742;
   1:L PR[91] R[100]mm/sec CNT100;
   1:  PR[91,1] = PR[90,1] + 14.527;
   1:  PR[91,2] = PR[90,2] + 19.315;
   1:L PR[91] R[100]mm/sec CNT100;
   1:  PR[91,1] = PR[90,1] + 9.836;
   1:  PR[91,2] = PR[90,2] + 18.951;
   1:L PR[91] R[100]mm/sec CNT100;
   1:  PR[91,1] = PR[90,1] + 5.363;
   1:  PR[91,2] = PR[90,2] + 17.644;
   1:L PR[91] R[100]mm/sec CNT100;
   1:  PR[91,1] = PR[90,1] + 4.771;
   1:  PR[91,2] = PR[90,2] + 17.345;
   1:L PR[91] R[100]mm/sec CNT100;
   1:  PR[91,1] = PR[90,1] + 1.938;
   1:  PR[91,2] = PR[90,2] + 15.796;
   1:L PR[91] R[100]mm/sec CNT100;
   1:  PR[91,1] = PR[90,1] + 1.434;
   1:  PR[91,2] = PR[90,2] + 15.436;
   1:L PR[91] R[100]mm/sec CNT100;
   1:  PR[91,1] = PR[90,1] + 0.367;
   1:  PR[91,2] = PR[90,2] + 15.273;
   1:L PR[91] R[100]mm/sec CNT100;
   1:  PR[91,1] = PR[90,1] + -0.302;
   1:  PR[91,2] = PR[90,2] + 15.040;
   1:L PR[91] R[100]mm/sec CNT100;
   1:  PR[91] = PR[90];
   1:  PR[91,1] = PR[90,1] + -2.076;
   1:  PR[91,2] = PR[90,2] + 16.111;
   1:  PR[91,3] = PR[90,3] + 39.195;
   1:L PR[91] R[100]mm/sec CNT100;
   1:  PR[91,1] = PR[90,1] + -3.718;
   1:  PR[91,2] = PR[90,2] + 17.010;
   1:L PR[91] R[100]mm/sec CNT100;
   1:  PR[91,1] = PR[90,1] + -5.377;
   1:  PR[91,2] = PR[90,2] + 17.850;
   1:L PR[91] R[100]mm/sec CNT100;
   1:  PR[91,1] = PR[90,1] + -9.457;
   1:  PR[91,2] = PR[90,2] + 19.043;
   1:L PR[91] R[100]mm/sec CNT100;
   1:  PR[91,1] = PR[90,1] + -9.837;
   1:  PR[91,2] = PR[90,2] + 19.143;
   1:L PR[91] R[100]mm/sec CNT100;
   1:  PR[91,1] = PR[90,1] + -14.504;
   1:  PR[91,2] = PR[90,2] + 19.459;
   1:L PR[91] R[100]mm/sec CNT100;
   1:  PR[91,1] = PR[90,1] + -16.542;
   1:  PR[91,2] = PR[90,2] + 19.165;
   1:L PR[91] R[100]mm/sec CNT100;
   1:  PR[91,1] = PR[90,1] + -19.162;
   1:  PR[91,2] = PR[90,2] + 18.817;
   1:L PR[91] R[100]mm/sec CNT100;
   1:  PR[91,1] = PR[90,1] + -23.567;
   1:  PR[91,2] = PR[90,2] + 17.229;
   1:L PR[91] R[100]mm/sec CNT100;
   1:  PR[91,1] = PR[90,1] + -23.706;
   1:  PR[91,2] = PR[90,2] + 17.153;
   1:L PR[91] R[100]mm/sec CNT100;
   1:  PR[91,1] = PR[90,1] + -27.242;
   1:  PR[91,2] = PR[90,2] + 14.950;
   1:L PR[91] R[100]mm/sec CNT100;
   1:  PR[91,1] = PR[90,1] + -27.520;
   1:  PR[91,2] = PR[90,2] + 14.745;
   1:L PR[91] R[100]mm/sec CNT100;
   1:  PR[91,1] = PR[90,1] + -30.576;
   1:  PR[91,2] = PR[90,2] + 11.752;
   1:L PR[91] R[100]mm/sec CNT100;
   1:  PR[91,1] = PR[90,1] + -30.910;
   1:  PR[91,2] = PR[90,2] + 11.317;
   1:L PR[91] R[100]mm/sec CNT100;
   1:  PR[91,1] = PR[90,1] + -32.753;
   1:  PR[91,2] = PR[90,2] + 8.444;
   1:L PR[91] R[100]mm/sec CNT100;
   1:  PR[91,1] = PR[90,1] + -33.103;
   1:  PR[91,2] = PR[90,2] + 7.821;
   1:L PR[91] R[100]mm/sec CNT100;
   1:  PR[91,1] = PR[90,1] + -33.396;
   1:  PR[91,2] = PR[90,2] + 7.067;
   1:L PR[91] R[100]mm/sec CNT100;
   1:  PR[91,1] = PR[90,1] + -34.468;
   1:  PR[91,2] = PR[90,2] + 4.139;
   1:L PR[91] R[100]mm/sec CNT100;
   1:  PR[91,1] = PR[90,1] + -34.614;
   1:  PR[91,2] = PR[90,2] + 3.489;
   1:L PR[91] R[100]mm/sec CNT100;
   1:  PR[91,1] = PR[90,1] + -34.677;
   1:  PR[91,2] = PR[90,2] + 2.581;
   1:L PR[91] R[100]mm/sec CNT100;
   1:  PR[91,1] = PR[90,1] + -35.030;
   1:  PR[91,2] = PR[90,2] + -0.479;
   1:L PR[91] R[100]mm/sec CNT100;
   1:  PR[91,1] = PR[90,1] + -34.976;
   1:  PR[91,2] = PR[90,2] + -1.258;
   1:L PR[91] R[100]mm/sec CNT100;
   1:  PR[91,1] = PR[90,1] + -34.626;
   1:  PR[91,2] = PR[90,2] + -4.282;
   1:L PR[91] R[100]mm/sec CNT100;
   1:  PR[91,1] = PR[90,1] + -34.473;
   1:  PR[91,2] = PR[90,2] + -4.962;
   1:L PR[91] R[100]mm/sec CNT100;
   1:  PR[91,1] = PR[90,1] + -34.160;
   1:  PR[91,2] = PR[90,2] + -5.767;
   1:L PR[91] R[100]mm/sec CNT100;
   1:  PR[91,1] = PR[90,1] + -33.091;
   1:  PR[91,2] = PR[90,2] + -8.690;
   1:L PR[91] R[100]mm/sec CNT100;
   1:  PR[91,1] = PR[90,1] + -32.753;
   1:  PR[91,2] = PR[90,2] + -9.292;
   1:L PR[91] R[100]mm/sec CNT100;
   1:  PR[91,1] = PR[90,1] + -30.910;
   1:  PR[91,2] = PR[90,2] + -12.164;
   1:L PR[91] R[100]mm/sec CNT100;
   1:  PR[91,1] = PR[90,1] + -30.576;
   1:  PR[91,2] = PR[90,2] + -12.599;
   1:L PR[91] R[100]mm/sec CNT100;
   1:  PR[91,1] = PR[90,1] + -27.520;
   1:  PR[91,2] = PR[90,2] + -15.592;
   1:L PR[91] R[100]mm/sec CNT100;
   1:  PR[91,1] = PR[90,1] + -27.242;
   1:  PR[91,2] = PR[90,2] + -15.797;
   1:L PR[91] R[100]mm/sec CNT100;
   1:  PR[91,1] = PR[90,1] + -23.706;
   1:  PR[91,2] = PR[90,2] + -18.000;
   1:L PR[91] R[100]mm/sec CNT100;
   1:  PR[91,1] = PR[90,1] + -23.566;
   1:  PR[91,2] = PR[90,2] + -18.076;
   1:L PR[91] R[100]mm/sec CNT100;
   1:  PR[91,1] = PR[90,1] + -19.162;
   1:  PR[91,2] = PR[90,2] + -19.664;
   1:L PR[91] R[100]mm/sec CNT100;
   1:  PR[91,1] = PR[90,1] + -16.543;
   1:  PR[91,2] = PR[90,2] + -20.012;
   1:L PR[91] R[100]mm/sec CNT100;
   1:  PR[91,1] = PR[90,1] + -14.503;
   1:  PR[91,2] = PR[90,2] + -20.307;
   1:L PR[91] R[100]mm/sec CNT100;
   1:  PR[91,1] = PR[90,1] + -9.836;
   1:  PR[91,2] = PR[90,2] + -19.990;
   1:L PR[91] R[100]mm/sec CNT100;
   1:  PR[91,1] = PR[90,1] + -9.456;
   1:  PR[91,2] = PR[90,2] + -19.890;
   1:L PR[91] R[100]mm/sec CNT100;
   1:  PR[91,1] = PR[90,1] + -5.329;
   1:  PR[91,2] = PR[90,2] + -18.683;
   1:L PR[91] R[100]mm/sec CNT100;
   1:  PR[91,1] = PR[90,1] + -5.307;
   1:  PR[91,2] = PR[90,2] + -18.673;
   1:L PR[91] R[100]mm/sec CNT100;
   1:  PR[91,1] = PR[90,1] + -3.680;
   1:  PR[91,2] = PR[90,2] + -17.837;
   1:L PR[91] R[100]mm/sec CNT100;
   1:  PR[91,1] = PR[90,1] + -2.077;
   1:  PR[91,2] = PR[90,2] + -16.960;
   1:L PR[91] R[100]mm/sec CNT100;
   1:  PR[91,1] = PR[90,1] + -0.280;
   1:  PR[91,2] = PR[90,2] + -16.350;
   1:L PR[91] R[100]mm/sec CNT100;
   1:  PR[91,1] = PR[90,1] + 0.770;
   1:  PR[91,2] = PR[90,2] + -16.716;
   1:L PR[91] R[100]mm/sec CNT100;
   1:  PR[91,1] = PR[90,1] + 1.485;
   1:  PR[91,2] = PR[90,2] + -16.825;
   1:L PR[91] R[100]mm/sec CNT100;
   1:  PR[91,1] = PR[90,1] + 1.908;
   1:  PR[91,2] = PR[90,2] + -17.132;
   1:L PR[91] R[100]mm/sec CNT100;
   1:  PR[91,1] = PR[90,1] + 3.235;
   1:  PR[91,2] = PR[90,2] + -17.857;
   1:L PR[91] R[100]mm/sec CNT100;
   1:  PR[91,1] = PR[90,1] + 4.821;
   1:  PR[91,2] = PR[90,2] + -18.670;
   1:L PR[91] R[100]mm/sec CNT100;
   1:  PR[91,1] = PR[90,1] + 4.845;
   1:  PR[91,2] = PR[90,2] + -18.681;
   1:L PR[91] R[100]mm/sec CNT100;
   1:  PR[91,1] = PR[90,1] + 8.973;
   1:  PR[91,2] = PR[90,2] + -19.889;
   1:L PR[91] R[100]mm/sec CNT100;
   1:  PR[91,1] = PR[90,1] + 9.353;
   1:  PR[91,2] = PR[90,2] + -19.988;
   1:L PR[91] R[100]mm/sec CNT100;
   1:  PR[91,1] = PR[90,1] + 14.020;
   1:  PR[91,2] = PR[90,2] + -20.307;
   1:L PR[91] R[100]mm/sec CNT100;
   1:  PR[91,1] = PR[90,1] + 16.062;
   1:  PR[91,2] = PR[90,2] + -20.012;
   1:L PR[91] R[100]mm/sec CNT100;
   1:  PR[91,1] = PR[90,1] + 18.678;
   1:  PR[91,2] = PR[90,2] + -19.664;
   1:L PR[91] R[100]mm/sec CNT100;
   1:  PR[91,1] = PR[90,1] + 23.085;
   1:  PR[91,2] = PR[90,2] + -18.077;
   1:L PR[91] R[100]mm/sec CNT100;
   1:  PR[91,1] = PR[90,1] + 23.223;
   1:  PR[91,2] = PR[90,2] + -18.002;
   1:L PR[91] R[100]mm/sec CNT100;
   1:  PR[91,1] = PR[90,1] + 26.758;
   1:  PR[91,2] = PR[90,2] + -15.803;
   1:L PR[91] R[100]mm/sec CNT100;
   1:  PR[91,1] = PR[90,1] + 27.029;
   1:  PR[91,2] = PR[90,2] + -15.604;
   1:L PR[91] R[100]mm/sec CNT100;
   1:  PR[91,1] = PR[90,1] + 30.084;
   1:  PR[91,2] = PR[90,2] + -12.608;
   1:L PR[91] R[100]mm/sec CNT100;
   1:  PR[91,1] = PR[90,1] + 30.423;
   1:  PR[91,2] = PR[90,2] + -12.167;
   1:L PR[91] R[100]mm/sec CNT100;
   1:  PR[91,1] = PR[90,1] + 32.268;
   1:  PR[91,2] = PR[90,2] + -9.295;
   1:L PR[91] R[100]mm/sec CNT100;
   1:  PR[91,1] = PR[90,1] + 32.623;
   1:  PR[91,2] = PR[90,2] + -8.669;
   1:L PR[91] R[100]mm/sec CNT100;
   1:  PR[91,1] = PR[90,1] + 32.912;
   1:  PR[91,2] = PR[90,2] + -7.935;
   1:L PR[91] R[100]mm/sec CNT100;
   1:  PR[91,1] = PR[90,1] + 33.983;
   1:  PR[91,2] = PR[90,2] + -5.021;
   1:L PR[91] R[100]mm/sec CNT100;
   1:  PR[91,1] = PR[90,1] + 34.130;
   1:  PR[91,2] = PR[90,2] + -4.376;
   1:L PR[91] R[100]mm/sec CNT100;
   1:  PR[91,1] = PR[90,1] + 34.197;
   1:  PR[91,2] = PR[90,2] + -3.439;
   1:L PR[91] R[100]mm/sec CNT100;
   1:  PR[91,1] = PR[90,1] + 34.550;
   1:  PR[91,2] = PR[90,2] + -0.371;
   1:L PR[91] R[100]mm/sec CNT100;
   1:  PR[91,1] = PR[90,1] + 34.492;
   1:  PR[91,2] = PR[90,2] + 0.443;
   1:L PR[91] R[100]mm/sec CNT100;
   1:  PR[91,1] = PR[90,1] + 34.142;
   1:  PR[91,2] = PR[90,2] + 3.477;
   1:L PR[91] R[100]mm/sec CNT100;
   1:  PR[91,1] = PR[90,1] + 33.990;
   1:  PR[91,2] = PR[90,2] + 4.146;
   1:L PR[91] R[100]mm/sec CNT100;
   1:  PR[91,1] = PR[90,1] + 33.678;
   1:  PR[91,2] = PR[90,2] + 4.936;
   1:L PR[91] R[100]mm/sec CNT100;
   1:  PR[91,1] = PR[90,1] + 32.609;
   1:  PR[91,2] = PR[90,2] + 7.846;
   1:L PR[91] R[100]mm/sec CNT100;
   1:  PR[91,1] = PR[90,1] + 32.268;
   1:  PR[91,2] = PR[90,2] + 8.448;
   1:L PR[91] R[100]mm/sec CNT100;
   1:  PR[91,1] = PR[90,1] + 30.423;
   1:  PR[91,2] = PR[90,2] + 11.319;
   1:L PR[91] R[100]mm/sec CNT100;
   1:  PR[91,1] = PR[90,1] + 30.084;
   1:  PR[91,2] = PR[90,2] + 11.760;
   1:L PR[91] R[100]mm/sec CNT100;
   1:  PR[91,1] = PR[90,1] + 27.029;
   1:  PR[91,2] = PR[90,2] + 14.757;
   1:L PR[91] R[100]mm/sec CNT100;
   1:  PR[91,1] = PR[90,1] + 26.758;
   1:  PR[91,2] = PR[90,2] + 14.956;
   1:L PR[91] R[100]mm/sec CNT100;
   1:  PR[91,1] = PR[90,1] + 23.223;
   1:  PR[91,2] = PR[90,2] + 17.155;
   1:L PR[91] R[100]mm/sec CNT100;
   1:  PR[91,1] = PR[90,1] + 23.067;
   1:  PR[91,2] = PR[90,2] + 17.240;
   1:L PR[91] R[100]mm/sec CNT100;
   1:  PR[91,1] = PR[90,1] + 22.898;
   1:  PR[91,2] = PR[90,2] + 17.304;
   1:L PR[91] R[100]mm/sec CNT100;
   1:  PR[91,1] = PR[90,1] + 18.679;
   1:  PR[91,2] = PR[90,2] + 18.817;
   1:L PR[91] R[100]mm/sec CNT100;
   1:  PR[91,1] = PR[90,1] + 16.062;
   1:  PR[91,2] = PR[90,2] + 19.165;
   1:L PR[91] R[100]mm/sec CNT100;
   1:  PR[91,1] = PR[90,1] + 14.021;
   1:  PR[91,2] = PR[90,2] + 19.460;
   1:L PR[91] R[100]mm/sec CNT100;
   1:  PR[91,1] = PR[90,1] + 9.353;
   1:  PR[91,2] = PR[90,2] + 19.141;
   1:L PR[91] R[100]mm/sec CNT100;
   1:  PR[91,1] = PR[90,1] + 8.974;
   1:  PR[91,2] = PR[90,2] + 19.042;
   1:L PR[91] R[100]mm/sec CNT100;
   1:  PR[91,1] = PR[90,1] + 4.892;
   1:  PR[91,2] = PR[90,2] + 17.848;
   1:L PR[91] R[100]mm/sec CNT100;
   1:  PR[91,1] = PR[90,1] + 3.243;
   1:  PR[91,2] = PR[90,2] + 17.014;
   1:L PR[91] R[100]mm/sec CNT100;
   1:  PR[91,1] = PR[90,1] + 1.901;
   1:  PR[91,2] = PR[90,2] + 16.280;
   1:L PR[91] R[100]mm/sec CNT100;
   1:  PR[91,1] = PR[90,1] + 1.474;
   1:  PR[91,2] = PR[90,2] + 15.975;
   1:L PR[91] R[100]mm/sec CNT100;
   1:  PR[91,1] = PR[90,1] + 0.765;
   1:  PR[91,2] = PR[90,2] + 15.867;
   1:L PR[91] R[100]mm/sec CNT100;
   1:  PR[91,1] = PR[90,1] + -0.280;
   1:  PR[91,2] = PR[90,2] + 15.503;
   1:L PR[91] R[100]mm/sec CNT100;
   1:  PR[91] = PR[90];
   1:  PR[91,1] = PR[90,1] + -2.025;
   1:  PR[91,2] = PR[90,2] + 16.594;
   1:  PR[91,3] = PR[90,3] + 40.495;
   1:L PR[91] R[100]mm/sec CNT100;
   1:  PR[91,1] = PR[90,1] + -4.725;
   1:  PR[91,2] = PR[90,2] + 17.979;
   1:L PR[91] R[100]mm/sec CNT100;
   1:  PR[91,1] = PR[90,1] + -4.857;
   1:  PR[91,2] = PR[90,2] + 18.039;
   1:L PR[91] R[100]mm/sec CNT100;
   1:  PR[91,1] = PR[90,1] + -8.429;
   1:  PR[91,2] = PR[90,2] + 19.084;
   1:L PR[91] R[100]mm/sec CNT100;
   1:  PR[91,1] = PR[90,1] + -9.399;
   1:  PR[91,2] = PR[90,2] + 19.338;
   1:L PR[91] R[100]mm/sec CNT100;
   1:  PR[91,1] = PR[90,1] + -13.509;
   1:  PR[91,2] = PR[90,2] + 19.622;
   1:L PR[91] R[100]mm/sec CNT100;
   1:  PR[91,1] = PR[90,1] + -14.054;
   1:  PR[91,2] = PR[90,2] + 19.644;
   1:L PR[91] R[100]mm/sec CNT100;
   1:  PR[91,1] = PR[90,1] + -18.704;
   1:  PR[91,2] = PR[90,2] + 18.964;
   1:L PR[91] R[100]mm/sec CNT100;
   1:  PR[91,1] = PR[90,1] + -23.069;
   1:  PR[91,2] = PR[90,2] + 17.352;
   1:L PR[91] R[100]mm/sec CNT100;
   1:  PR[91,1] = PR[90,1] + -26.990;
   1:  PR[91,2] = PR[90,2] + 14.912;
   1:L PR[91] R[100]mm/sec CNT100;
   1:  PR[91,1] = PR[90,1] + -30.212;
   1:  PR[91,2] = PR[90,2] + 11.754;
   1:L PR[91] R[100]mm/sec CNT100;
   1:  PR[91,1] = PR[90,1] + -30.325;
   1:  PR[91,2] = PR[90,2] + 11.607;
   1:L PR[91] R[100]mm/sec CNT100;
   1:  PR[91,1] = PR[90,1] + -32.487;
   1:  PR[91,2] = PR[90,2] + 8.236;
   1:L PR[91] R[100]mm/sec CNT100;
   1:  PR[91,1] = PR[90,1] + -32.661;
   1:  PR[91,2] = PR[90,2] + 7.928;
   1:L PR[91] R[100]mm/sec CNT100;
   1:  PR[91,1] = PR[90,1] + -32.817;
   1:  PR[91,2] = PR[90,2] + 7.527;
   1:L PR[91] R[100]mm/sec CNT100;
   1:  PR[91,1] = PR[90,1] + -34.093;
   1:  PR[91,2] = PR[90,2] + 4.041;
   1:L PR[91] R[100]mm/sec CNT100;
   1:  PR[91,1] = PR[90,1] + -34.163;
   1:  PR[91,2] = PR[90,2] + 3.730;
   1:L PR[91] R[100]mm/sec CNT100;
   1:  PR[91,1] = PR[90,1] + -34.201;
   1:  PR[91,2] = PR[90,2] + 3.180;
   1:L PR[91] R[100]mm/sec CNT100;
   1:  PR[91,1] = PR[90,1] + -34.623;
   1:  PR[91,2] = PR[90,2] + -0.479;
   1:L PR[91] R[100]mm/sec CNT100;
   1:  PR[91,1] = PR[90,1] + -34.593;
   1:  PR[91,2] = PR[90,2] + -0.908;
   1:L PR[91] R[100]mm/sec CNT100;
   1:  PR[91,1] = PR[90,1] + -34.175;
   1:  PR[91,2] = PR[90,2] + -4.523;
   1:L PR[91] R[100]mm/sec CNT100;
   1:  PR[91,1] = PR[90,1] + -34.098;
   1:  PR[91,2] = PR[90,2] + -4.864;
   1:L PR[91] R[100]mm/sec CNT100;
   1:  PR[91,1] = PR[90,1] + -33.913;
   1:  PR[91,2] = PR[90,2] + -5.339;
   1:L PR[91] R[100]mm/sec CNT100;
   1:  PR[91,1] = PR[90,1] + -32.649;
   1:  PR[91,2] = PR[90,2] + -8.796;
   1:L PR[91] R[100]mm/sec CNT100;
   1:  PR[91,1] = PR[90,1] + -32.487;
   1:  PR[91,2] = PR[90,2] + -9.084;
   1:L PR[91] R[100]mm/sec CNT100;
   1:  PR[91,1] = PR[90,1] + -30.325;
   1:  PR[91,2] = PR[90,2] + -12.455;
   1:L PR[91] R[100]mm/sec CNT100;
   1:  PR[91,1] = PR[90,1] + -30.212;
   1:  PR[91,2] = PR[90,2] + -12.602;
   1:L PR[91] R[100]mm/sec CNT100;
   1:  PR[91,1] = PR[90,1] + -26.990;
   1:  PR[91,2] = PR[90,2] + -15.759;
   1:L PR[91] R[100]mm/sec CNT100;
   1:  PR[91,1] = PR[90,1] + -23.069;
   1:  PR[91,2] = PR[90,2] + -18.199;
   1:L PR[91] R[100]mm/sec CNT100;
   1:  PR[91,1] = PR[90,1] + -18.703;
   1:  PR[91,2] = PR[90,2] + -19.811;
   1:L PR[91] R[100]mm/sec CNT100;
   1:  PR[91,1] = PR[90,1] + -14.054;
   1:  PR[91,2] = PR[90,2] + -20.491;
   1:L PR[91] R[100]mm/sec CNT100;
   1:  PR[91,1] = PR[90,1] + -13.509;
   1:  PR[91,2] = PR[90,2] + -20.469;
   1:L PR[91] R[100]mm/sec CNT100;
   1:  PR[91,1] = PR[90,1] + -9.399;
   1:  PR[91,2] = PR[90,2] + -20.185;
   1:L PR[91] R[100]mm/sec CNT100;
   1:  PR[91,1] = PR[90,1] + -8.428;
   1:  PR[91,2] = PR[90,2] + -19.931;
   1:L PR[91] R[100]mm/sec CNT100;
   1:  PR[91,1] = PR[90,1] + -4.857;
   1:  PR[91,2] = PR[90,2] + -18.886;
   1:L PR[91] R[100]mm/sec CNT100;
   1:  PR[91,1] = PR[90,1] + -4.706;
   1:  PR[91,2] = PR[90,2] + -18.817;
   1:L PR[91] R[100]mm/sec CNT100;
   1:  PR[91,1] = PR[90,1] + -2.024;
   1:  PR[91,2] = PR[90,2] + -17.439;
   1:L PR[91] R[100]mm/sec CNT100;
   1:  PR[91,1] = PR[90,1] + -0.255;
   1:  PR[91,2] = PR[90,2] + -16.814;
   1:L PR[91] R[100]mm/sec CNT100;
   1:  PR[91,1] = PR[90,1] + 1.534;
   1:  PR[91,2] = PR[90,2] + -17.437;
   1:L PR[91] R[100]mm/sec CNT100;
   1:  PR[91,1] = PR[90,1] + 4.221;
   1:  PR[91,2] = PR[90,2] + -18.815;
   1:L PR[91] R[100]mm/sec CNT100;
   1:  PR[91,1] = PR[90,1] + 4.374;
   1:  PR[91,2] = PR[90,2] + -18.885;
   1:L PR[91] R[100]mm/sec CNT100;
   1:  PR[91,1] = PR[90,1] + 7.945;
   1:  PR[91,2] = PR[90,2] + -19.929;
   1:L PR[91] R[100]mm/sec CNT100;
   1:  PR[91,1] = PR[90,1] + 8.916;
   1:  PR[91,2] = PR[90,2] + -20.184;
   1:L PR[91] R[100]mm/sec CNT100;
   1:  PR[91,1] = PR[90,1] + 13.027;
   1:  PR[91,2] = PR[90,2] + -20.469;
   1:L PR[91] R[100]mm/sec CNT100;
   1:  PR[91,1] = PR[90,1] + 13.571;
   1:  PR[91,2] = PR[90,2] + -20.492;
   1:L PR[91] R[100]mm/sec CNT100;
   1:  PR[91,1] = PR[90,1] + 18.221;
   1:  PR[91,2] = PR[90,2] + -19.811;
   1:L PR[91] R[100]mm/sec CNT100;
   1:  PR[91,1] = PR[90,1] + 22.588;
   1:  PR[91,2] = PR[90,2] + -18.200;
   1:L PR[91] R[100]mm/sec CNT100;
   1:  PR[91,1] = PR[90,1] + 26.506;
   1:  PR[91,2] = PR[90,2] + -15.765;
   1:L PR[91] R[100]mm/sec CNT100;
   1:  PR[91,1] = PR[90,1] + 29.724;
   1:  PR[91,2] = PR[90,2] + -12.604;
   1:L PR[91] R[100]mm/sec CNT100;
   1:  PR[91,1] = PR[90,1] + 29.841;
   1:  PR[91,2] = PR[90,2] + -12.452;
   1:L PR[91] R[100]mm/sec CNT100;
   1:  PR[91,1] = PR[90,1] + 32.005;
   1:  PR[91,2] = PR[90,2] + -9.084;
   1:L PR[91] R[100]mm/sec CNT100;
   1:  PR[91,1] = PR[90,1] + 32.182;
   1:  PR[91,2] = PR[90,2] + -8.772;
   1:L PR[91] R[100]mm/sec CNT100;
   1:  PR[91,1] = PR[90,1] + 32.335;
   1:  PR[91,2] = PR[90,2] + -8.384;
   1:L PR[91] R[100]mm/sec CNT100;
   1:  PR[91,1] = PR[90,1] + 33.610;
   1:  PR[91,2] = PR[90,2] + -4.915;
   1:L PR[91] R[100]mm/sec CNT100;
   1:  PR[91,1] = PR[90,1] + 33.680;
   1:  PR[91,2] = PR[90,2] + -4.607;
   1:L PR[91] R[100]mm/sec CNT100;
   1:  PR[91,1] = PR[90,1] + 33.721;
   1:  PR[91,2] = PR[90,2] + -4.040;
   1:L PR[91] R[100]mm/sec CNT100;
   1:  PR[91,1] = PR[90,1] + 34.143;
   1:  PR[91,2] = PR[90,2] + -0.371;
   1:L PR[91] R[100]mm/sec CNT100;
   1:  PR[91,1] = PR[90,1] + 34.111;
   1:  PR[91,2] = PR[90,2] + 0.082;
   1:L PR[91] R[100]mm/sec CNT100;
   1:  PR[91,1] = PR[90,1] + 33.692;
   1:  PR[91,2] = PR[90,2] + 3.709;
   1:L PR[91] R[100]mm/sec CNT100;
   1:  PR[91,1] = PR[90,1] + 33.617;
   1:  PR[91,2] = PR[90,2] + 4.040;
   1:L PR[91] R[100]mm/sec CNT100;
   1:  PR[91,1] = PR[90,1] + 33.432;
   1:  PR[91,2] = PR[90,2] + 4.507;
   1:L PR[91] R[100]mm/sec CNT100;
   1:  PR[91,1] = PR[90,1] + 32.168;
   1:  PR[91,2] = PR[90,2] + 7.949;
   1:L PR[91] R[100]mm/sec CNT100;
   1:  PR[91,1] = PR[90,1] + 32.005;
   1:  PR[91,2] = PR[90,2] + 8.237;
   1:L PR[91] R[100]mm/sec CNT100;
   1:  PR[91,1] = PR[90,1] + 29.841;
   1:  PR[91,2] = PR[90,2] + 11.605;
   1:L PR[91] R[100]mm/sec CNT100;
   1:  PR[91,1] = PR[90,1] + 29.724;
   1:  PR[91,2] = PR[90,2] + 11.757;
   1:L PR[91] R[100]mm/sec CNT100;
   1:  PR[91,1] = PR[90,1] + 26.506;
   1:  PR[91,2] = PR[90,2] + 14.918;
   1:L PR[91] R[100]mm/sec CNT100;
   1:  PR[91,1] = PR[90,1] + 22.588;
   1:  PR[91,2] = PR[90,2] + 17.352;
   1:L PR[91] R[100]mm/sec CNT100;
   1:  PR[91,1] = PR[90,1] + 18.221;
   1:  PR[91,2] = PR[90,2] + 18.964;
   1:L PR[91] R[100]mm/sec CNT100;
   1:  PR[91,1] = PR[90,1] + 13.571;
   1:  PR[91,2] = PR[90,2] + 19.645;
   1:L PR[91] R[100]mm/sec CNT100;
   1:  PR[91,1] = PR[90,1] + 13.027;
   1:  PR[91,2] = PR[90,2] + 19.622;
   1:L PR[91] R[100]mm/sec CNT100;
   1:  PR[91,1] = PR[90,1] + 8.917;
   1:  PR[91,2] = PR[90,2] + 19.337;
   1:L PR[91] R[100]mm/sec CNT100;
   1:  PR[91,1] = PR[90,1] + 7.946;
   1:  PR[91,2] = PR[90,2] + 19.082;
   1:L PR[91] R[100]mm/sec CNT100;
   1:  PR[91,1] = PR[90,1] + 4.374;
   1:  PR[91,2] = PR[90,2] + 18.037;
   1:L PR[91] R[100]mm/sec CNT100;
   1:  PR[91,1] = PR[90,1] + 4.240;
   1:  PR[91,2] = PR[90,2] + 17.976;
   1:L PR[91] R[100]mm/sec CNT100;
   1:  PR[91,1] = PR[90,1] + 1.530;
   1:  PR[91,2] = PR[90,2] + 16.589;
   1:L PR[91] R[100]mm/sec CNT100;
   1:  PR[91,1] = PR[90,1] + -0.258;
   1:  PR[91,2] = PR[90,2] + 15.966;
   1:L PR[91] R[100]mm/sec CNT100;
   1:  PR[91] = PR[90];
   1:  PR[91,1] = PR[90,1] + -1.438;
   1:  PR[91,2] = PR[90,2] + 16.869;
   1:  PR[91,3] = PR[90,3] + 41.795;
   1:L PR[91] R[100]mm/sec CNT100;
   1:  PR[91,1] = PR[90,1] + -1.781;
   1:  PR[91,2] = PR[90,2] + 16.921;
   1:L PR[91] R[100]mm/sec CNT100;
   1:  PR[91,1] = PR[90,1] + -4.131;
   1:  PR[91,2] = PR[90,2] + 18.127;
   1:L PR[91] R[100]mm/sec CNT100;
   1:  PR[91,1] = PR[90,1] + -4.386;
   1:  PR[91,2] = PR[90,2] + 18.243;
   1:L PR[91] R[100]mm/sec CNT100;
   1:  PR[91,1] = PR[90,1] + -7.401;
   1:  PR[91,2] = PR[90,2] + 19.124;
   1:L PR[91] R[100]mm/sec CNT100;
   1:  PR[91,1] = PR[90,1] + -8.961;
   1:  PR[91,2] = PR[90,2] + 19.534;
   1:L PR[91] R[100]mm/sec CNT100;
   1:  PR[91,1] = PR[90,1] + -12.491;
   1:  PR[91,2] = PR[90,2] + 19.777;
   1:L PR[91] R[100]mm/sec CNT100;
   1:  PR[91,1] = PR[90,1] + -13.641;
   1:  PR[91,2] = PR[90,2] + 19.824;
   1:L PR[91] R[100]mm/sec CNT100;
   1:  PR[91,1] = PR[90,1] + -17.559;
   1:  PR[91,2] = PR[90,2] + 19.259;
   1:L PR[91] R[100]mm/sec CNT100;
   1:  PR[91,1] = PR[90,1] + -18.279;
   1:  PR[91,2] = PR[90,2] + 19.136;
   1:L PR[91] R[100]mm/sec CNT100;
   1:  PR[91,1] = PR[90,1] + -22.359;
   1:  PR[91,2] = PR[90,2] + 17.621;
   1:L PR[91] R[100]mm/sec CNT100;
   1:  PR[91,1] = PR[90,1] + -22.645;
   1:  PR[91,2] = PR[90,2] + 17.507;
   1:L PR[91] R[100]mm/sec CNT100;
   1:  PR[91,1] = PR[90,1] + -26.550;
   1:  PR[91,2] = PR[90,2] + 15.015;
   1:L PR[91] R[100]mm/sec CNT100;
   1:  PR[91,1] = PR[90,1] + -28.204;
   1:  PR[91,2] = PR[90,2] + 13.368;
   1:L PR[91] R[100]mm/sec CNT100;
   1:  PR[91,1] = PR[90,1] + -29.776;
   1:  PR[91,2] = PR[90,2] + 11.827;
   1:L PR[91] R[100]mm/sec CNT100;
   1:  PR[91,1] = PR[90,1] + -32.210;
   1:  PR[91,2] = PR[90,2] + 8.046;
   1:L PR[91] R[100]mm/sec CNT100;
   1:  PR[91,1] = PR[90,1] + -33.712;
   1:  PR[91,2] = PR[90,2] + 3.956;
   1:L PR[91] R[100]mm/sec CNT100;
   1:  PR[91,1] = PR[90,1] + -33.725;
   1:  PR[91,2] = PR[90,2] + 3.779;
   1:L PR[91] R[100]mm/sec CNT100;
   1:  PR[91,1] = PR[90,1] + -34.216;
   1:  PR[91,2] = PR[90,2] + -0.479;
   1:L PR[91] R[100]mm/sec CNT100;
   1:  PR[91,1] = PR[90,1] + -34.210;
   1:  PR[91,2] = PR[90,2] + -0.558;
   1:L PR[91] R[100]mm/sec CNT100;
   1:  PR[91,1] = PR[90,1] + -33.723;
   1:  PR[91,2] = PR[90,2] + -4.764;
   1:L PR[91] R[100]mm/sec CNT100;
   1:  PR[91,1] = PR[90,1] + -33.666;
   1:  PR[91,2] = PR[90,2] + -4.912;
   1:L PR[91] R[100]mm/sec CNT100;
   1:  PR[91,1] = PR[90,1] + -32.209;
   1:  PR[91,2] = PR[90,2] + -8.895;
   1:L PR[91] R[100]mm/sec CNT100;
   1:  PR[91,1] = PR[90,1] + -29.776;
   1:  PR[91,2] = PR[90,2] + -12.674;
   1:L PR[91] R[100]mm/sec CNT100;
   1:  PR[91,1] = PR[90,1] + -28.204;
   1:  PR[91,2] = PR[90,2] + -14.215;
   1:L PR[91] R[100]mm/sec CNT100;
   1:  PR[91,1] = PR[90,1] + -26.550;
   1:  PR[91,2] = PR[90,2] + -15.863;
   1:L PR[91] R[100]mm/sec CNT100;
   1:  PR[91,1] = PR[90,1] + -22.645;
   1:  PR[91,2] = PR[90,2] + -18.355;
   1:L PR[91] R[100]mm/sec CNT100;
   1:  PR[91,1] = PR[90,1] + -22.359;
   1:  PR[91,2] = PR[90,2] + -18.469;
   1:L PR[91] R[100]mm/sec CNT100;
   1:  PR[91,1] = PR[90,1] + -18.278;
   1:  PR[91,2] = PR[90,2] + -19.983;
   1:L PR[91] R[100]mm/sec CNT100;
   1:  PR[91,1] = PR[90,1] + -17.558;
   1:  PR[91,2] = PR[90,2] + -20.106;
   1:L PR[91] R[100]mm/sec CNT100;
   1:  PR[91,1] = PR[90,1] + -13.641;
   1:  PR[91,2] = PR[90,2] + -20.672;
   1:L PR[91] R[100]mm/sec CNT100;
   1:  PR[91,1] = PR[90,1] + -12.490;
   1:  PR[91,2] = PR[90,2] + -20.624;
   1:L PR[91] R[100]mm/sec CNT100;
   1:  PR[91,1] = PR[90,1] + -8.960;
   1:  PR[91,2] = PR[90,2] + -20.381;
   1:L PR[91] R[100]mm/sec CNT100;
   1:  PR[91,1] = PR[90,1] + -7.399;
   1:  PR[91,2] = PR[90,2] + -19.971;
   1:L PR[91] R[100]mm/sec CNT100;
   1:  PR[91,1] = PR[90,1] + -4.385;
   1:  PR[91,2] = PR[90,2] + -19.090;
   1:L PR[91] R[100]mm/sec CNT100;
   1:  PR[91,1] = PR[90,1] + -4.105;
   1:  PR[91,2] = PR[90,2] + -18.962;
   1:L PR[91] R[100]mm/sec CNT100;
   1:  PR[91,1] = PR[90,1] + -1.784;
   1:  PR[91,2] = PR[90,2] + -17.769;
   1:L PR[91] R[100]mm/sec CNT100;
   1:  PR[91,1] = PR[90,1] + -1.434;
   1:  PR[91,2] = PR[90,2] + -17.715;
   1:L PR[91] R[100]mm/sec CNT100;
   1:  PR[91,1] = PR[90,1] + -0.229;
   1:  PR[91,2] = PR[90,2] + -17.287;
   1:L PR[91] R[100]mm/sec CNT100;
   1:  PR[91,1] = PR[90,1] + 1.487;
   1:  PR[91,2] = PR[90,2] + -17.866;
   1:L PR[91] R[100]mm/sec CNT100;
   1:  PR[91,1] = PR[90,1] + 3.621;
   1:  PR[91,2] = PR[90,2] + -18.960;
   1:L PR[91] R[100]mm/sec CNT100;
   1:  PR[91,1] = PR[90,1] + 3.903;
   1:  PR[91,2] = PR[90,2] + -19.088;
   1:L PR[91] R[100]mm/sec CNT100;
   1:  PR[91,1] = PR[90,1] + 6.917;
   1:  PR[91,2] = PR[90,2] + -19.970;
   1:L PR[91] R[100]mm/sec CNT100;
   1:  PR[91,1] = PR[90,1] + 8.478;
   1:  PR[91,2] = PR[90,2] + -20.380;
   1:L PR[91] R[100]mm/sec CNT100;
   1:  PR[91,1] = PR[90,1] + 12.008;
   1:  PR[91,2] = PR[90,2] + -20.625;
   1:L PR[91] R[100]mm/sec CNT100;
   1:  PR[91,1] = PR[90,1] + 13.158;
   1:  PR[91,2] = PR[90,2] + -20.672;
   1:L PR[91] R[100]mm/sec CNT100;
   1:  PR[91,1] = PR[90,1] + 17.075;
   1:  PR[91,2] = PR[90,2] + -20.106;
   1:L PR[91] R[100]mm/sec CNT100;
   1:  PR[91,1] = PR[90,1] + 17.796;
   1:  PR[91,2] = PR[90,2] + -19.983;
   1:L PR[91] R[100]mm/sec CNT100;
   1:  PR[91,1] = PR[90,1] + 21.878;
   1:  PR[91,2] = PR[90,2] + -18.469;
   1:L PR[91] R[100]mm/sec CNT100;
   1:  PR[91,1] = PR[90,1] + 22.165;
   1:  PR[91,2] = PR[90,2] + -18.355;
   1:L PR[91] R[100]mm/sec CNT100;
   1:  PR[91,1] = PR[90,1] + 26.055;
   1:  PR[91,2] = PR[90,2] + -15.880;
   1:L PR[91] R[100]mm/sec CNT100;
   1:  PR[91,1] = PR[90,1] + 27.721;
   1:  PR[91,2] = PR[90,2] + -14.216;
   1:L PR[91] R[100]mm/sec CNT100;
   1:  PR[91,1] = PR[90,1] + 29.318;
   1:  PR[91,2] = PR[90,2] + -12.647;
   1:L PR[91] R[100]mm/sec CNT100;
   1:  PR[91,1] = PR[90,1] + 31.731;
   1:  PR[91,2] = PR[90,2] + -8.891;
   1:L PR[91] R[100]mm/sec CNT100;
   1:  PR[91,1] = PR[90,1] + 33.232;
   1:  PR[91,2] = PR[90,2] + -4.824;
   1:L PR[91] R[100]mm/sec CNT100;
   1:  PR[91,1] = PR[90,1] + 33.245;
   1:  PR[91,2] = PR[90,2] + -4.641;
   1:L PR[91] R[100]mm/sec CNT100;
   1:  PR[91,1] = PR[90,1] + 33.736;
   1:  PR[91,2] = PR[90,2] + -0.371;
   1:L PR[91] R[100]mm/sec CNT100;
   1:  PR[91,1] = PR[90,1] + 33.729;
   1:  PR[91,2] = PR[90,2] + -0.279;
   1:L PR[91] R[100]mm/sec CNT100;
   1:  PR[91,1] = PR[90,1] + 33.242;
   1:  PR[91,2] = PR[90,2] + 3.940;
   1:L PR[91] R[100]mm/sec CNT100;
   1:  PR[91,1] = PR[90,1] + 33.238;
   1:  PR[91,2] = PR[90,2] + 3.961;
   1:L PR[91] R[100]mm/sec CNT100;
   1:  PR[91,1] = PR[90,1] + 31.731;
   1:  PR[91,2] = PR[90,2] + 8.043;
   1:L PR[91] R[100]mm/sec CNT100;
   1:  PR[91,1] = PR[90,1] + 29.293;
   1:  PR[91,2] = PR[90,2] + 11.823;
   1:L PR[91] R[100]mm/sec CNT100;
   1:  PR[91,1] = PR[90,1] + 27.721;
   1:  PR[91,2] = PR[90,2] + 13.369;
   1:L PR[91] R[100]mm/sec CNT100;
   1:  PR[91,1] = PR[90,1] + 26.056;
   1:  PR[91,2] = PR[90,2] + 15.032;
   1:L PR[91] R[100]mm/sec CNT100;
   1:  PR[91,1] = PR[90,1] + 22.165;
   1:  PR[91,2] = PR[90,2] + 17.508;
   1:L PR[91] R[100]mm/sec CNT100;
   1:  PR[91,1] = PR[90,1] + 21.878;
   1:  PR[91,2] = PR[90,2] + 17.622;
   1:L PR[91] R[100]mm/sec CNT100;
   1:  PR[91,1] = PR[90,1] + 17.796;
   1:  PR[91,2] = PR[90,2] + 19.135;
   1:L PR[91] R[100]mm/sec CNT100;
   1:  PR[91,1] = PR[90,1] + 17.075;
   1:  PR[91,2] = PR[90,2] + 19.259;
   1:L PR[91] R[100]mm/sec CNT100;
   1:  PR[91,1] = PR[90,1] + 13.158;
   1:  PR[91,2] = PR[90,2] + 19.825;
   1:L PR[91] R[100]mm/sec CNT100;
   1:  PR[91,1] = PR[90,1] + 12.008;
   1:  PR[91,2] = PR[90,2] + 19.777;
   1:L PR[91] R[100]mm/sec CNT100;
   1:  PR[91,1] = PR[90,1] + 8.479;
   1:  PR[91,2] = PR[90,2] + 19.533;
   1:L PR[91] R[100]mm/sec CNT100;
   1:  PR[91,1] = PR[90,1] + 6.919;
   1:  PR[91,2] = PR[90,2] + 19.123;
   1:L PR[91] R[100]mm/sec CNT100;
   1:  PR[91,1] = PR[90,1] + 3.903;
   1:  PR[91,2] = PR[90,2] + 18.241;
   1:L PR[91] R[100]mm/sec CNT100;
   1:  PR[91,1] = PR[90,1] + 3.647;
   1:  PR[91,2] = PR[90,2] + 18.125;
   1:L PR[91] R[100]mm/sec CNT100;
   1:  PR[91,1] = PR[90,1] + 1.486;
   1:  PR[91,2] = PR[90,2] + 17.018;
   1:L PR[91] R[100]mm/sec CNT100;
   1:  PR[91,1] = PR[90,1] + -0.230;
   1:  PR[91,2] = PR[90,2] + 16.440;
   1:L PR[91] R[100]mm/sec CNT100;
   1:  PR[91] = PR[90];
   1:  PR[91,1] = PR[90,1] + -1.219;
   1:  PR[91,2] = PR[90,2] + 17.275;
   1:  PR[91,3] = PR[90,3] + 43.095;
   1:L PR[91] R[100]mm/sec CNT100;
   1:  PR[91,1] = PR[90,1] + -1.745;
   1:  PR[91,2] = PR[90,2] + 17.355;
   1:L PR[91] R[100]mm/sec CNT100;
   1:  PR[91,1] = PR[90,1] + -3.537;
   1:  PR[91,2] = PR[90,2] + 18.275;
   1:L PR[91] R[100]mm/sec CNT100;
   1:  PR[91,1] = PR[90,1] + -3.914;
   1:  PR[91,2] = PR[90,2] + 18.446;
   1:L PR[91] R[100]mm/sec CNT100;
   1:  PR[91,1] = PR[90,1] + -6.372;
   1:  PR[91,2] = PR[90,2] + 19.165;
   1:L PR[91] R[100]mm/sec CNT100;
   1:  PR[91,1] = PR[90,1] + -8.522;
   1:  PR[91,2] = PR[90,2] + 19.729;
   1:L PR[91] R[100]mm/sec CNT100;
   1:  PR[91,1] = PR[90,1] + -11.472;
   1:  PR[91,2] = PR[90,2] + 19.932;
   1:L PR[91] R[100]mm/sec CNT100;
   1:  PR[91,1] = PR[90,1] + -13.226;
   1:  PR[91,2] = PR[90,2] + 20.005;
   1:L PR[91] R[100]mm/sec CNT100;
   1:  PR[91,1] = PR[90,1] + -16.552;
   1:  PR[91,2] = PR[90,2] + 19.524;
   1:L PR[91] R[100]mm/sec CNT100;
   1:  PR[91,1] = PR[90,1] + -17.883;
   1:  PR[91,2] = PR[90,2] + 19.297;
   1:L PR[91] R[100]mm/sec CNT100;
   1:  PR[91,1] = PR[90,1] + -21.392;
   1:  PR[91,2] = PR[90,2] + 17.995;
   1:L PR[91] R[100]mm/sec CNT100;
   1:  PR[91,1] = PR[90,1] + -22.266;
   1:  PR[91,2] = PR[90,2] + 17.646;
   1:L PR[91] R[100]mm/sec CNT100;
   1:  PR[91,1] = PR[90,1] + -25.707;
   1:  PR[91,2] = PR[90,2] + 15.454;
   1:L PR[91] R[100]mm/sec CNT100;
   1:  PR[91,1] = PR[90,1] + -26.164;
   1:  PR[91,2] = PR[90,2] + 15.148;
   1:L PR[91] R[100]mm/sec CNT100;
   1:  PR[91,1] = PR[90,1] + -29.245;
   1:  PR[91,2] = PR[90,2] + 12.079;
   1:L PR[91] R[100]mm/sec CNT100;
   1:  PR[91,1] = PR[90,1] + -29.390;
   1:  PR[91,2] = PR[90,2] + 11.928;
   1:L PR[91] R[100]mm/sec CNT100;
   1:  PR[91,1] = PR[90,1] + -31.815;
   1:  PR[91,2] = PR[90,2] + 8.091;
   1:L PR[91] R[100]mm/sec CNT100;
   1:  PR[91,1] = PR[90,1] + -33.300;
   1:  PR[91,2] = PR[90,2] + 3.984;
   1:L PR[91] R[100]mm/sec CNT100;
   1:  PR[91,1] = PR[90,1] + -33.803;
   1:  PR[91,2] = PR[90,2] + -0.424;
   1:L PR[91] R[100]mm/sec CNT100;
   1:  PR[91,1] = PR[90,1] + -33.300;
   1:  PR[91,2] = PR[90,2] + -4.831;
   1:L PR[91] R[100]mm/sec CNT100;
   1:  PR[91,1] = PR[90,1] + -31.815;
   1:  PR[91,2] = PR[90,2] + -8.938;
   1:L PR[91] R[100]mm/sec CNT100;
   1:  PR[91,1] = PR[90,1] + -29.402;
   1:  PR[91,2] = PR[90,2] + -12.757;
   1:L PR[91] R[100]mm/sec CNT100;
   1:  PR[91,1] = PR[90,1] + -26.161;
   1:  PR[91,2] = PR[90,2] + -15.997;
   1:L PR[91] R[100]mm/sec CNT100;
   1:  PR[91,1] = PR[90,1] + -25.707;
   1:  PR[91,2] = PR[90,2] + -16.301;
   1:L PR[91] R[100]mm/sec CNT100;
   1:  PR[91,1] = PR[90,1] + -22.265;
   1:  PR[91,2] = PR[90,2] + -18.494;
   1:L PR[91] R[100]mm/sec CNT100;
   1:  PR[91,1] = PR[90,1] + -21.392;
   1:  PR[91,2] = PR[90,2] + -18.842;
   1:L PR[91] R[100]mm/sec CNT100;
   1:  PR[91,1] = PR[90,1] + -17.882;
   1:  PR[91,2] = PR[90,2] + -20.144;
   1:L PR[91] R[100]mm/sec CNT100;
   1:  PR[91,1] = PR[90,1] + -16.551;
   1:  PR[91,2] = PR[90,2] + -20.372;
   1:L PR[91] R[100]mm/sec CNT100;
   1:  PR[91,1] = PR[90,1] + -13.225;
   1:  PR[91,2] = PR[90,2] + -20.852;
   1:L PR[91] R[100]mm/sec CNT100;
   1:  PR[91,1] = PR[90,1] + -11.471;
   1:  PR[91,2] = PR[90,2] + -20.780;
   1:L PR[91] R[100]mm/sec CNT100;
   1:  PR[91,1] = PR[90,1] + -8.522;
   1:  PR[91,2] = PR[90,2] + -20.576;
   1:L PR[91] R[100]mm/sec CNT100;
   1:  PR[91,1] = PR[90,1] + -6.370;
   1:  PR[91,2] = PR[90,2] + -20.011;
   1:L PR[91] R[100]mm/sec CNT100;
   1:  PR[91,1] = PR[90,1] + -3.914;
   1:  PR[91,2] = PR[90,2] + -19.293;
   1:L PR[91] R[100]mm/sec CNT100;
   1:  PR[91,1] = PR[90,1] + -3.504;
   1:  PR[91,2] = PR[90,2] + -19.106;
   1:L PR[91] R[100]mm/sec CNT100;
   1:  PR[91,1] = PR[90,1] + -1.748;
   1:  PR[91,2] = PR[90,2] + -18.204;
   1:L PR[91] R[100]mm/sec CNT100;
   1:  PR[91,1] = PR[90,1] + -1.216;
   1:  PR[91,2] = PR[90,2] + -18.122;
   1:L PR[91] R[100]mm/sec CNT100;
   1:  PR[91,1] = PR[90,1] + -0.175;
   1:  PR[91,2] = PR[90,2] + -17.752;
   1:L PR[91] R[100]mm/sec CNT100;
   1:  PR[91,1] = PR[90,1] + 1.011;
   1:  PR[91,2] = PR[90,2] + -18.165;
   1:L PR[91] R[100]mm/sec CNT100;
   1:  PR[91,1] = PR[90,1] + 1.382;
   1:  PR[91,2] = PR[90,2] + -18.265;
   1:L PR[91] R[100]mm/sec CNT100;
   1:  PR[91,1] = PR[90,1] + 3.021;
   1:  PR[91,2] = PR[90,2] + -19.104;
   1:L PR[91] R[100]mm/sec CNT100;
   1:  PR[91,1] = PR[90,1] + 3.432;
   1:  PR[91,2] = PR[90,2] + -19.292;
   1:L PR[91] R[100]mm/sec CNT100;
   1:  PR[91,1] = PR[90,1] + 5.889;
   1:  PR[91,2] = PR[90,2] + -20.011;
   1:L PR[91] R[100]mm/sec CNT100;
   1:  PR[91,1] = PR[90,1] + 8.040;
   1:  PR[91,2] = PR[90,2] + -20.575;
   1:L PR[91] R[100]mm/sec CNT100;
   1:  PR[91,1] = PR[90,1] + 10.990;
   1:  PR[91,2] = PR[90,2] + -20.780;
   1:L PR[91] R[100]mm/sec CNT100;
   1:  PR[91,1] = PR[90,1] + 12.743;
   1:  PR[91,2] = PR[90,2] + -20.852;
   1:L PR[91] R[100]mm/sec CNT100;
   1:  PR[91,1] = PR[90,1] + 16.069;
   1:  PR[91,2] = PR[90,2] + -20.372;
   1:L PR[91] R[100]mm/sec CNT100;
   1:  PR[91,1] = PR[90,1] + 17.401;
   1:  PR[91,2] = PR[90,2] + -20.144;
   1:L PR[91] R[100]mm/sec CNT100;
   1:  PR[91,1] = PR[90,1] + 20.911;
   1:  PR[91,2] = PR[90,2] + -18.843;
   1:L PR[91] R[100]mm/sec CNT100;
   1:  PR[91,1] = PR[90,1] + 21.785;
   1:  PR[91,2] = PR[90,2] + -18.494;
   1:L PR[91] R[100]mm/sec CNT100;
   1:  PR[91,1] = PR[90,1] + 25.226;
   1:  PR[91,2] = PR[90,2] + -16.305;
   1:L PR[91] R[100]mm/sec CNT100;
   1:  PR[91,1] = PR[90,1] + 25.679;
   1:  PR[91,2] = PR[90,2] + -16.002;
   1:L PR[91] R[100]mm/sec CNT100;
   1:  PR[91,1] = PR[90,1] + 28.921;
   1:  PR[91,2] = PR[90,2] + -12.752;
   1:L PR[91] R[100]mm/sec CNT100;
   1:  PR[91,1] = PR[90,1] + 31.336;
   1:  PR[91,2] = PR[90,2] + -8.935;
   1:L PR[91] R[100]mm/sec CNT100;
   1:  PR[91,1] = PR[90,1] + 32.820;
   1:  PR[91,2] = PR[90,2] + -4.849;
   1:L PR[91] R[100]mm/sec CNT100;
   1:  PR[91,1] = PR[90,1] + 33.323;
   1:  PR[91,2] = PR[90,2] + -0.424;
   1:L PR[91] R[100]mm/sec CNT100;
   1:  PR[91,1] = PR[90,1] + 32.820;
   1:  PR[91,2] = PR[90,2] + 4.001;
   1:L PR[91] R[100]mm/sec CNT100;
   1:  PR[91,1] = PR[90,1] + 31.336;
   1:  PR[91,2] = PR[90,2] + 8.088;
   1:L PR[91] R[100]mm/sec CNT100;
   1:  PR[91,1] = PR[90,1] + 28.921;
   1:  PR[91,2] = PR[90,2] + 11.905;
   1:L PR[91] R[100]mm/sec CNT100;
   1:  PR[91,1] = PR[90,1] + 25.679;
   1:  PR[91,2] = PR[90,2] + 15.155;
   1:L PR[91] R[100]mm/sec CNT100;
   1:  PR[91,1] = PR[90,1] + 25.226;
   1:  PR[91,2] = PR[90,2] + 15.458;
   1:L PR[91] R[100]mm/sec CNT100;
   1:  PR[91,1] = PR[90,1] + 21.785;
   1:  PR[91,2] = PR[90,2] + 17.647;
   1:L PR[91] R[100]mm/sec CNT100;
   1:  PR[91,1] = PR[90,1] + 20.911;
   1:  PR[91,2] = PR[90,2] + 17.995;
   1:L PR[91] R[100]mm/sec CNT100;
   1:  PR[91,1] = PR[90,1] + 17.401;
   1:  PR[91,2] = PR[90,2] + 19.297;
   1:L PR[91] R[100]mm/sec CNT100;
   1:  PR[91,1] = PR[90,1] + 16.069;
   1:  PR[91,2] = PR[90,2] + 19.524;
   1:L PR[91] R[100]mm/sec CNT100;
   1:  PR[91,1] = PR[90,1] + 12.743;
   1:  PR[91,2] = PR[90,2] + 20.005;
   1:L PR[91] R[100]mm/sec CNT100;
   1:  PR[91,1] = PR[90,1] + 10.990;
   1:  PR[91,2] = PR[90,2] + 19.933;
   1:L PR[91] R[100]mm/sec CNT100;
   1:  PR[91,1] = PR[90,1] + 8.041;
   1:  PR[91,2] = PR[90,2] + 19.728;
   1:L PR[91] R[100]mm/sec CNT100;
   1:  PR[91,1] = PR[90,1] + 5.891;
   1:  PR[91,2] = PR[90,2] + 19.164;
   1:L PR[91] R[100]mm/sec CNT100;
   1:  PR[91,1] = PR[90,1] + 3.432;
   1:  PR[91,2] = PR[90,2] + 18.445;
   1:L PR[91] R[100]mm/sec CNT100;
   1:  PR[91,1] = PR[90,1] + 3.054;
   1:  PR[91,2] = PR[90,2] + 18.273;
   1:L PR[91] R[100]mm/sec CNT100;
   1:  PR[91,1] = PR[90,1] + 1.377;
   1:  PR[91,2] = PR[90,2] + 17.414;
   1:L PR[91] R[100]mm/sec CNT100;
   1:  PR[91,1] = PR[90,1] + 1.007;
   1:  PR[91,2] = PR[90,2] + 17.317;
   1:L PR[91] R[100]mm/sec CNT100;
   1:  PR[91,1] = PR[90,1] + -0.176;
   1:  PR[91,2] = PR[90,2] + 16.905;
   1:L PR[91] R[100]mm/sec CNT100;
   1:  PR[91] = PR[90];
   1:  PR[91,1] = PR[90,1] + -1.000;
   1:  PR[91,2] = PR[90,2] + 17.682;
   1:  PR[91,3] = PR[90,3] + 44.395;
   1:L PR[91] R[100]mm/sec CNT100;
   1:  PR[91,1] = PR[90,1] + -1.709;
   1:  PR[91,2] = PR[90,2] + 17.789;
   1:L PR[91] R[100]mm/sec CNT100;
   1:  PR[91,1] = PR[90,1] + -2.943;
   1:  PR[91,2] = PR[90,2] + 18.422;
   1:L PR[91] R[100]mm/sec CNT100;
   1:  PR[91,1] = PR[90,1] + -3.443;
   1:  PR[91,2] = PR[90,2] + 18.650;
   1:L PR[91] R[100]mm/sec CNT100;
   1:  PR[91,1] = PR[90,1] + -5.344;
   1:  PR[91,2] = PR[90,2] + 19.206;
   1:L PR[91] R[100]mm/sec CNT100;
   1:  PR[91,1] = PR[90,1] + -8.083;
   1:  PR[91,2] = PR[90,2] + 19.924;
   1:L PR[91] R[100]mm/sec CNT100;
   1:  PR[91,1] = PR[90,1] + -10.453;
   1:  PR[91,2] = PR[90,2] + 20.088;
   1:L PR[91] R[100]mm/sec CNT100;
   1:  PR[91,1] = PR[90,1] + -12.810;
   1:  PR[91,2] = PR[90,2] + 20.185;
   1:L PR[91] R[100]mm/sec CNT100;
   1:  PR[91,1] = PR[90,1] + -15.544;
   1:  PR[91,2] = PR[90,2] + 19.790;
   1:L PR[91] R[100]mm/sec CNT100;
   1:  PR[91,1] = PR[90,1] + -17.487;
   1:  PR[91,2] = PR[90,2] + 19.458;
   1:L PR[91] R[100]mm/sec CNT100;
   1:  PR[91,1] = PR[90,1] + -20.425;
   1:  PR[91,2] = PR[90,2] + 18.368;
   1:L PR[91] R[100]mm/sec CNT100;
   1:  PR[91,1] = PR[90,1] + -21.885;
   1:  PR[91,2] = PR[90,2] + 17.786;
   1:L PR[91] R[100]mm/sec CNT100;
   1:  PR[91,1] = PR[90,1] + -24.807;
   1:  PR[91,2] = PR[90,2] + 15.924;
   1:L PR[91] R[100]mm/sec CNT100;
   1:  PR[91,1] = PR[90,1] + -25.795;
   1:  PR[91,2] = PR[90,2] + 15.263;
   1:L PR[91] R[100]mm/sec CNT100;
   1:  PR[91,1] = PR[90,1] + -28.439;
   1:  PR[91,2] = PR[90,2] + 12.630;
   1:L PR[91] R[100]mm/sec CNT100;
   1:  PR[91,1] = PR[90,1] + -29.032;
   1:  PR[91,2] = PR[90,2] + 12.015;
   1:L PR[91] R[100]mm/sec CNT100;
   1:  PR[91,1] = PR[90,1] + -31.138;
   1:  PR[91,2] = PR[90,2] + 8.686;
   1:L PR[91] R[100]mm/sec CNT100;
   1:  PR[91,1] = PR[90,1] + -31.455;
   1:  PR[91,2] = PR[90,2] + 8.168;
   1:L PR[91] R[100]mm/sec CNT100;
   1:  PR[91,1] = PR[90,1] + -32.951;
   1:  PR[91,2] = PR[90,2] + 4.014;
   1:L PR[91] R[100]mm/sec CNT100;
   1:  PR[91,1] = PR[90,1] + -33.412;
   1:  PR[91,2] = PR[90,2] + -0.035;
   1:L PR[91] R[100]mm/sec CNT100;
   1:  PR[91,1] = PR[90,1] + -33.440;
   1:  PR[91,2] = PR[90,2] + -0.384;
   1:L PR[91] R[100]mm/sec CNT100;
   1:  PR[91,1] = PR[90,1] + -33.094;
   1:  PR[91,2] = PR[90,2] + -3.407;
   1:L PR[91] R[100]mm/sec CNT100;
   1:  PR[91,1] = PR[90,1] + -32.944;
   1:  PR[91,2] = PR[90,2] + -4.888;
   1:L PR[91] R[100]mm/sec CNT100;
   1:  PR[91,1] = PR[90,1] + -32.812;
   1:  PR[91,2] = PR[90,2] + -5.269;
   1:L PR[91] R[100]mm/sec CNT100;
   1:  PR[91,1] = PR[90,1] + -31.456;
   1:  PR[91,2] = PR[90,2] + -9.014;
   1:L PR[91] R[100]mm/sec CNT100;
   1:  PR[91,1] = PR[90,1] + -31.138;
   1:  PR[91,2] = PR[90,2] + -9.533;
   1:L PR[91] R[100]mm/sec CNT100;
   1:  PR[91,1] = PR[90,1] + -29.031;
   1:  PR[91,2] = PR[90,2] + -12.863;
   1:L PR[91] R[100]mm/sec CNT100;
   1:  PR[91,1] = PR[90,1] + -28.439;
   1:  PR[91,2] = PR[90,2] + -13.477;
   1:L PR[91] R[100]mm/sec CNT100;
   1:  PR[91,1] = PR[90,1] + -25.795;
   1:  PR[91,2] = PR[90,2] + -16.110;
   1:L PR[91] R[100]mm/sec CNT100;
   1:  PR[91,1] = PR[90,1] + -24.807;
   1:  PR[91,2] = PR[90,2] + -16.772;
   1:L PR[91] R[100]mm/sec CNT100;
   1:  PR[91,1] = PR[90,1] + -21.885;
   1:  PR[91,2] = PR[90,2] + -18.633;
   1:L PR[91] R[100]mm/sec CNT100;
   1:  PR[91,1] = PR[90,1] + -20.424;
   1:  PR[91,2] = PR[90,2] + -19.215;
   1:L PR[91] R[100]mm/sec CNT100;
   1:  PR[91,1] = PR[90,1] + -17.486;
   1:  PR[91,2] = PR[90,2] + -20.306;
   1:L PR[91] R[100]mm/sec CNT100;
   1:  PR[91,1] = PR[90,1] + -15.544;
   1:  PR[91,2] = PR[90,2] + -20.637;
   1:L PR[91] R[100]mm/sec CNT100;
   1:  PR[91,1] = PR[90,1] + -12.810;
   1:  PR[91,2] = PR[90,2] + -21.032;
   1:L PR[91] R[100]mm/sec CNT100;
   1:  PR[91,1] = PR[90,1] + -10.453;
   1:  PR[91,2] = PR[90,2] + -20.935;
   1:L PR[91] R[100]mm/sec CNT100;
   1:  PR[91,1] = PR[90,1] + -8.083;
   1:  PR[91,2] = PR[90,2] + -20.771;
   1:L PR[91] R[100]mm/sec CNT100;
   1:  PR[91,1] = PR[90,1] + -5.341;
   1:  PR[91,2] = PR[90,2] + -20.052;
   1:L PR[91] R[100]mm/sec CNT100;
   1:  PR[91,1] = PR[90,1] + -3.442;
   1:  PR[91,2] = PR[90,2] + -19.497;
   1:L PR[91] R[100]mm/sec CNT100;
   1:  PR[91,1] = PR[90,1] + -2.904;
   1:  PR[91,2] = PR[90,2] + -19.251;
   1:L PR[91] R[100]mm/sec CNT100;
   1:  PR[91,1] = PR[90,1] + -1.712;
   1:  PR[91,2] = PR[90,2] + -18.638;
   1:L PR[91] R[100]mm/sec CNT100;
   1:  PR[91,1] = PR[90,1] + -0.999;
   1:  PR[91,2] = PR[90,2] + -18.529;
   1:L PR[91] R[100]mm/sec CNT100;
   1:  PR[91,1] = PR[90,1] + -0.134;
   1:  PR[91,2] = PR[90,2] + -18.221;
   1:L PR[91] R[100]mm/sec CNT100;
   1:  PR[91,1] = PR[90,1] + 0.871;
   1:  PR[91,2] = PR[90,2] + -18.572;
   1:L PR[91] R[100]mm/sec CNT100;
   1:  PR[91,1] = PR[90,1] + 1.347;
   1:  PR[91,2] = PR[90,2] + -18.699;
   1:L PR[91] R[100]mm/sec CNT100;
   1:  PR[91,1] = PR[90,1] + 2.420;
   1:  PR[91,2] = PR[90,2] + -19.249;
   1:L PR[91] R[100]mm/sec CNT100;
   1:  PR[91,1] = PR[90,1] + 2.961;
   1:  PR[91,2] = PR[90,2] + -19.495;
   1:L PR[91] R[100]mm/sec CNT100;
   1:  PR[91,1] = PR[90,1] + 4.861;
   1:  PR[91,2] = PR[90,2] + -20.051;
   1:L PR[91] R[100]mm/sec CNT100;
   1:  PR[91,1] = PR[90,1] + 7.602;
   1:  PR[91,2] = PR[90,2] + -20.771;
   1:L PR[91] R[100]mm/sec CNT100;
   1:  PR[91,1] = PR[90,1] + 9.972;
   1:  PR[91,2] = PR[90,2] + -20.935;
   1:L PR[91] R[100]mm/sec CNT100;
   1:  PR[91,1] = PR[90,1] + 12.328;
   1:  PR[91,2] = PR[90,2] + -21.032;
   1:L PR[91] R[100]mm/sec CNT100;
   1:  PR[91,1] = PR[90,1] + 15.062;
   1:  PR[91,2] = PR[90,2] + -20.637;
   1:L PR[91] R[100]mm/sec CNT100;
   1:  PR[91,1] = PR[90,1] + 17.005;
   1:  PR[91,2] = PR[90,2] + -20.305;
   1:L PR[91] R[100]mm/sec CNT100;
   1:  PR[91,1] = PR[90,1] + 19.943;
   1:  PR[91,2] = PR[90,2] + -19.216;
   1:L PR[91] R[100]mm/sec CNT100;
   1:  PR[91,1] = PR[90,1] + 21.405;
   1:  PR[91,2] = PR[90,2] + -18.634;
   1:L PR[91] R[100]mm/sec CNT100;
   1:  PR[91,1] = PR[90,1] + 24.326;
   1:  PR[91,2] = PR[90,2] + -16.775;
   1:L PR[91] R[100]mm/sec CNT100;
   1:  PR[91,1] = PR[90,1] + 25.313;
   1:  PR[91,2] = PR[90,2] + -16.115;
